LIN {X 0,Y 467.56,Z 130.239,A -85,B 0,C 180,E1 -7430.853,E2 -7430.853} C_VEL
LIN {X 0,Y 467.558,Z 130.24,A -85,B 0,C 180,E1 -7434.261,E2 -7434.261} C_VEL
LIN {X 0,Y 467.578,Z 130.242,A -85,B 0,C 180,E1 -7437.321,E2 -7437.321} C_VEL
LIN {X 0,Y 467.568,Z 130.238,A -85,B 0,C 180,E1 -7440.667,E2 -7440.667} C_VEL
LIN {X 0,Y 467.616,Z 130.238,A -85,B 0,C 180,E1 -7443.199,E2 -7443.199} C_VEL
LIN {X 0,Y 467.592,Z 130.235,A -85,B 0,C 180,E1 -7446.468,E2 -7446.468} C_VEL
LIN {X 0,Y 467.621,Z 130.233,A -85,B 0,C 180,E1 -7449.777,E2 -7449.777} C_VEL
LIN {X 0,Y 467.597,Z 130.235,A -85,B 0,C 180,E1 -7452.506,E2 -7452.506} C_VEL
LIN {X 0,Y 467.606,Z 130.241,A -85,B 0,C 180,E1 -7455.196,E2 -7455.196} C_VEL
LIN {X 0,Y 467.655,Z 130.228,A -85,B 0,C 180,E1 -7457.854,E2 -7457.854} C_VEL
LIN {X 0,Y 467.68,Z 130.228,A -85,B 0,C 180,E1 -7461.357,E2 -7461.357} C_VEL
LIN {X 0,Y 467.734,Z 130.217,A -85,B 0,C 180,E1 -7463.962,E2 -7463.962} C_VEL
LIN {X 0,Y 467.859,Z 130.204,A -85,B 0,C 180,E1 -7467.417,E2 -7467.417} C_VEL
LIN {X 0,Y 467.882,Z 130.199,A -85,B 0,C 180,E1 -7470,E2 -7470} C_VEL
LIN {X 0,Y 467.858,Z 130.208,A -85,B 0,C 180,E1 -7472.583,E2 -7472.583} C_VEL
LIN {X 0,Y 467.734,Z 130.218,A -85,B 0,C 180,E1 -7476.037,E2 -7476.037} C_VEL
LIN {X 0,Y 467.68,Z 130.232,A -85,B 0,C 180,E1 -7478.642,E2 -7478.642} C_VEL
LIN {X 0,Y 467.654,Z 130.23,A -85,B 0,C 180,E1 -7482.145,E2 -7482.145} C_VEL
LIN {X 0,Y 467.637,Z 130.23,A -85,B 0,C 180,E1 -7485.695,E2 -7485.695} C_VEL
LIN {X 0,Y 467.615,Z 130.236,A -85,B 0,C 180,E1 -7488.764,E2 -7488.764} C_VEL
LIN {X 0,Y 467.578,Z 130.237,A -85,B 0,C 180,E1 -7491.268,E2 -7491.268} C_VEL
LIN {X 0,Y 467.56,Z 130.243,A -85,B 0,C 180,E1 -7493.944,E2 -7493.944} C_VEL
LIN {X 0,Y 467.61,Z 130.234,A -85,B 0,C 180,E1 -7496.8,E2 -7496.8} C_VEL
LIN {X 0,Y 467.584,Z 130.239,A -85,B 0,C 180,E1 -7499.736,E2 -7499.736} C_VEL
LIN {X 0,Y 467.581,Z 130.238,A -85,B 0,C 180,E1 -7502.758,E2 -7502.758} C_VEL
LIN {X 0,Y 467.553,Z 130.246,A -85,B 0,C 180,E1 -7505.889,E2 -7505.889} C_VEL
LIN {X 0,Y 467.579,Z 130.237,A -85,B 0,C 180,E1 -7509.145,E2 -7509.145} C_VEL
LIN {X 0,Y 467.616,Z 130.233,A -85,B 0,C 180,E1 -7512.571,E2 -7512.571} C_VEL
LIN {X 0,Y 467.567,Z 130.239,A -85,B 0,C 180,E1 -7515.053,E2 -7515.053} C_VEL
LIN {X 0,Y 467.585,Z 130.24,A -85,B 0,C 180,E1 -7517.44,E2 -7517.44} C_VEL
LIN {X 0,Y 467.596,Z 130.235,A -85,B 0,C 180,E1 -7520.857,E2 -7520.857} C_VEL
LIN {X 0,Y 467.556,Z 130.241,A -85,B 0,C 180,E1 -7524.261,E2 -7524.261} C_VEL
LIN {X 0,Y 467.579,Z 130.241,A -85,B 0,C 180,E1 -7527.321,E2 -7527.321} C_VEL
LIN {X 0,Y 467.567,Z 130.238,A -85,B 0,C 180,E1 -7530.667,E2 -7530.667} C_VEL
LIN {X 0,Y 467.614,Z 130.237,A -85,B 0,C 180,E1 -7533.2,E2 -7533.2} C_VEL
LIN {X 0,Y 467.589,Z 130.236,A -85,B 0,C 180,E1 -7536.468,E2 -7536.468} C_VEL
LIN {X 0,Y 467.621,Z 130.234,A -85,B 0,C 180,E1 -7539.777,E2 -7539.777} C_VEL
LIN {X 0,Y 467.606,Z 130.234,A -85,B 0,C 180,E1 -7542.507,E2 -7542.507} C_VEL
LIN {X 0,Y 467.604,Z 130.242,A -85,B 0,C 180,E1 -7545.197,E2 -7545.197} C_VEL
LIN {X 0,Y 467.653,Z 130.228,A -85,B 0,C 180,E1 -7547.855,E2 -7547.855} C_VEL
LIN {X 0,Y 467.679,Z 130.228,A -85,B 0,C 180,E1 -7551.358,E2 -7551.358} C_VEL
LIN {X 0,Y 467.733,Z 130.218,A -85,B 0,C 180,E1 -7553.963,E2 -7553.963} C_VEL
LIN {X 0,Y 467.858,Z 130.204,A -85,B 0,C 180,E1 -7557.417,E2 -7557.417} C_VEL
LIN {X 0,Y 467.881,Z 130.199,A -85,B 0,C 180,E1 -7560,E2 -7560} C_VEL
LIN {X 0,Y 467.858,Z 130.207,A -85,B 0,C 180,E1 -7562.583,E2 -7562.583} C_VEL
LIN {X 0,Y 467.744,Z 130.217,A -85,B 0,C 180,E1 -7566.038,E2 -7566.038} C_VEL
LIN {X 0,Y 467.68,Z 130.232,A -85,B 0,C 180,E1 -7568.643,E2 -7568.643} C_VEL
LIN {X 0,Y 467.654,Z 130.23,A -85,B 0,C 180,E1 -7572.146,E2 -7572.146} C_VEL
LIN {X 0,Y 467.638,Z 130.23,A -85,B 0,C 180,E1 -7575.695,E2 -7575.695} C_VEL
LIN {X 0,Y 467.617,Z 130.236,A -85,B 0,C 180,E1 -7578.765,E2 -7578.765} C_VEL
LIN {X 0,Y 467.579,Z 130.237,A -85,B 0,C 180,E1 -7581.269,E2 -7581.269} C_VEL
LIN {X 0,Y 467.562,Z 130.242,A -85,B 0,C 180,E1 -7583.944,E2 -7583.944} C_VEL
LIN {X 0,Y 467.612,Z 130.235,A -85,B 0,C 180,E1 -7586.801,E2 -7586.801} C_VEL
LIN {X 0,Y 467.553,Z 130.242,A -85,B 0,C 180,E1 -7589.739,E2 -7589.739} C_VEL
LIN {X 0,Y 467.582,Z 130.238,A -85,B 0,C 180,E1 -7592.759,E2 -7592.759} C_VEL
LIN {X 0,Y 467.553,Z 130.245,A -85,B 0,C 180,E1 -7595.89,E2 -7595.89} C_VEL
LIN {X 0,Y 467.599,Z 130.234,A -85,B 0,C 180,E1 -7599.143,E2 -7599.143} C_VEL
LIN {X 0,Y 467.586,Z 130.237,A -85,B 0,C 180,E1 -7602.567,E2 -7602.567} C_VEL
LIN {X 0,Y 467.57,Z 130.238,A -85,B 0,C 180,E1 -7605.054,E2 -7605.054} C_VEL
LIN {X 0,Y 467.589,Z 130.238,A -85,B 0,C 180,E1 -7607.44,E2 -7607.44} C_VEL
LIN {X 0,Y 467.583,Z 130.236,A -85,B 0,C 180,E1 -7610.856,E2 -7610.856} C_VEL
LIN {X 0,Y 467.56,Z 130.241,A -85,B 0,C 180,E1 -7614.261,E2 -7614.261} C_VEL
LIN {X 0,Y 467.583,Z 130.24,A -85,B 0,C 180,E1 -7617.321,E2 -7617.321} C_VEL
LIN {X 0,Y 467.571,Z 130.239,A -85,B 0,C 180,E1 -7620.668,E2 -7620.668} C_VEL
LIN {X 0,Y 467.68,Z 130.252,A -85,B 0,C 180,E1 -7623.036,E2 -7623.036} C_VEL
LIN {X 0,Y 470.044,Z 142.535,A -85,B 0,C 180,E1 -7625.251,E2 -7625.251} C_VEL
LIN {X 0,Y 469.607,Z 155.018,A -85,B 0,C 180,E1 -7627.334,E2 -7627.334} C_VEL
LIN {X 0,Y 468.864,Z 174.362,A -85,B 0,C 180,E1 -7630.518,E2 -7630.518} C_VEL
LIN {X 0,Y 468.265,Z 190.123,A -85,B 0,C 180,E1 -7633.038,E2 -7633.038} C_VEL
LIN {X 0,Y 470.986,Z 210.09,A -85,B 0,C 180,E1 -7633.469,E2 -7633.469} C_VEL
LIN {X 0,Y 470.185,Z 299.083,A -85,B 0,C 180,E1 -7634.948,E2 -7634.948} C_VEL
LIN {X 0,Y 469.767,Z 311.954,A -85,B 0,C 180,E1 -7635.322,E2 -7635.322} C_VEL
LIN {X 0,Y 469.341,Z 324.553,A -85,B 0,C 180,E1 -7635.862,E2 -7635.862} C_VEL
LIN {X 0,Y 468.828,Z 336.62,A -85,B 0,C 180,E1 -7636.565,E2 -7636.565} C_VEL
LIN {X 0,Y 468.36,Z 347.957,A -85,B 0,C 180,E1 -7637.415,E2 -7637.415} C_VEL
LIN {X 0,Y 467.946,Z 358.612,A -85,B 0,C 180,E1 -7638.412,E2 -7638.412} C_VEL
LIN {X 0,Y 467.549,Z 367.139,A -85,B 0,C 180,E1 -7639.39,E2 -7639.39} C_VEL
LIN {X 0,Y 467.186,Z 376.379,A -85,B 0,C 180,E1 -7640.694,E2 -7640.694} C_VEL
LIN {X 0,Y 466.953,Z 383.82,A -85,B 0,C 180,E1 -7641.998,E2 -7641.998} C_VEL
LIN {X 0,Y 466.776,Z 389.92,A -85,B 0,C 180,E1 -7643.334,E2 -7643.334} C_VEL
LIN {X 0,Y 466.761,Z 395.107,A -85,B 0,C 180,E1 -7644.817,E2 -7644.817} C_VEL
LIN {X 0,Y 466.66,Z 397.46,A -85,B 0,C 180,E1 -7645.682,E2 -7645.682} C_VEL
LIN {X 0,Y 466.747,Z 399.385,A -85,B 0,C 180,E1 -7646.547,E2 -7646.547} C_VEL
LIN {X 0,Y 466.711,Z 400.833,A -85,B 0,C 180,E1 -7647.411,E2 -7647.411} C_VEL
LIN {X 0,Y 466.696,Z 401.849,A -85,B 0,C 180,E1 -7648.274,E2 -7648.274} C_VEL
LIN {X 0,Y 466.633,Z 402.462,A -85,B 0,C 180,E1 -7649.137,E2 -7649.137} C_VEL
LIN {X 0,Y 466.621,Z 402.677,A -85,B 0,C 180,E1 -7650,E2 -7650} C_VEL
LIN {X 0,Y 466.634,Z 402.447,A -85,B 0,C 180,E1 -7650.863,E2 -7650.863} C_VEL
LIN {X 0,Y 466.697,Z 401.808,A -85,B 0,C 180,E1 -7651.726,E2 -7651.726} C_VEL
LIN {X 0,Y 466.711,Z 400.765,A -85,B 0,C 180,E1 -7652.59,E2 -7652.59} C_VEL
LIN {X 0,Y 466.748,Z 399.31,A -85,B 0,C 180,E1 -7653.453,E2 -7653.453} C_VEL
LIN {X 0,Y 466.691,Z 396.254,A -85,B 0,C 180,E1 -7654.751,E2 -7654.751} C_VEL
LIN {X 0,Y 466.711,Z 392.13,A -85,B 0,C 180,E1 -7656.051,E2 -7656.051} C_VEL
LIN {X 0,Y 466.893,Z 385.791,A -85,B 0,C 180,E1 -7657.569,E2 -7657.569} C_VEL
LIN {X 0,Y 467.066,Z 378.887,A -85,B 0,C 180,E1 -7658.873,E2 -7658.873} C_VEL
LIN {X 0,Y 467.372,Z 370.326,A -85,B 0,C 180,E1 -7660.177,E2 -7660.177} C_VEL
LIN {X 0,Y 467.793,Z 361.513,A -85,B 0,C 180,E1 -7661.263,E2 -7661.263} C_VEL
LIN {X 0,Y 468.178,Z 351.631,A -85,B 0,C 180,E1 -7662.264,E2 -7662.264} C_VEL
LIN {X 0,Y 468.717,Z 339.929,A -85,B 0,C 180,E1 -7663.219,E2 -7663.219} C_VEL
LIN {X 0,Y 469.256,Z 327.977,A -85,B 0,C 180,E1 -7663.976,E2 -7663.976} C_VEL
LIN {X 0,Y 469.729,Z 315.638,A -85,B 0,C 180,E1 -7664.569,E2 -7664.569} C_VEL
LIN {X 0,Y 470.081,Z 304.036,A -85,B 0,C 180,E1 -7664.973,E2 -7664.973} C_VEL
LIN {X 0,Y 470.398,Z 290.664,A -85,B 0,C 180,E1 -7665.268,E2 -7665.268} C_VEL
LIN {X 0,Y 471.065,Z 208.796,A -85,B 0,C 180,E1 -7666.64,E2 -7666.64} C_VEL
LIN {X 0,Y 468.218,Z 188.105,A -85,B 0,C 180,E1 -7667.129,E2 -7667.129} C_VEL
LIN {X 0,Y 468.776,Z 170.52,A -85,B 0,C 180,E1 -7669.943,E2 -7669.943} C_VEL
LIN {X 0,Y 469.353,Z 153.611,A -85,B 0,C 180,E1 -7672.68,E2 -7672.68} C_VEL
LIN {X 0,Y 469.853,Z 142.026,A -85,B 0,C 180,E1 -7674.571,E2 -7674.571} C_VEL
LIN {X 0,Y 468.115,Z 132.345,A -85,B 0,C 180,E1 -7676.289,E2 -7676.289} C_VEL
LIN {X 0,Y 467.659,Z 130.236,A -85,B 0,C 180,E1 -7676.677,E2 -7676.677} C_VEL
LIN {X 0,Y 467.558,Z 130.25,A -85,B 0,C 180,E1 -7679.738,E2 -7679.738} C_VEL
LIN {X 0,Y 467.587,Z 130.241,A -85,B 0,C 180,E1 -7682.758,E2 -7682.758} C_VEL
LIN {X 0,Y 467.557,Z 130.246,A -85,B 0,C 180,E1 -7685.89,E2 -7685.89} C_VEL
LIN {X 0,Y 467.586,Z 130.239,A -85,B 0,C 180,E1 -7689.145,E2 -7689.145} C_VEL
LIN {X 0,Y 467.59,Z 130.239,A -85,B 0,C 180,E1 -7692.567,E2 -7692.567} C_VEL
LIN {X 0,Y 467.574,Z 130.239,A -85,B 0,C 180,E1 -7695.053,E2 -7695.053} C_VEL
LIN {X 0,Y 467.592,Z 130.239,A -85,B 0,C 180,E1 -7697.44,E2 -7697.44} C_VEL
LIN {X 0,Y 467.563,Z 130.237,A -85,B 0,C 180,E1 -7700.853,E2 -7700.853} C_VEL
LIN {X 0,Y 467.562,Z 130.239,A -85,B 0,C 180,E1 -7704.261,E2 -7704.261} C_VEL
LIN {X 0,Y 467.582,Z 130.241,A -85,B 0,C 180,E1 -7707.321,E2 -7707.321} C_VEL
LIN {X 0,Y 467.572,Z 130.239,A -85,B 0,C 180,E1 -7710.668,E2 -7710.668} C_VEL
LIN {X 0,Y 467.619,Z 130.24,A -85,B 0,C 180,E1 -7713.2,E2 -7713.2} C_VEL
LIN {X 0,Y 467.596,Z 130.236,A -85,B 0,C 180,E1 -7716.468,E2 -7716.468} C_VEL
LIN {X 0,Y 467.625,Z 130.232,A -85,B 0,C 180,E1 -7719.777,E2 -7719.777} C_VEL
LIN {X 0,Y 467.598,Z 130.235,A -85,B 0,C 180,E1 -7722.506,E2 -7722.506} C_VEL
LIN {X 0,Y 467.607,Z 130.24,A -85,B 0,C 180,E1 -7725.196,E2 -7725.196} C_VEL
LIN {X 0,Y 467.659,Z 130.229,A -85,B 0,C 180,E1 -7727.854,E2 -7727.854} C_VEL
LIN {X 0,Y 467.672,Z 130.23,A -85,B 0,C 180,E1 -7731.357,E2 -7731.357} C_VEL
LIN {X 0,Y 467.726,Z 130.223,A -85,B 0,C 180,E1 -7733.962,E2 -7733.962} C_VEL
LIN {X 0,Y 467.854,Z 130.207,A -85,B 0,C 180,E1 -7737.417,E2 -7737.417} C_VEL
LIN {X 0,Y 467.882,Z 130.204,A -85,B 0,C 180,E1 -7740,E2 -7740} C_VEL
LIN {X 0,Y 467.849,Z 130.212,A -85,B 0,C 180,E1 -7742.583,E2 -7742.583} C_VEL
LIN {X 0,Y 467.745,Z 130.412,A -85,B 0,C 180,E1 -7745.55,E2 -7745.55} C_VEL
LIN {X 0,Y 468.818,Z 136.804,A -85,B 0,C 180,E1 -7746.891,E2 -7746.891} C_VEL
LIN {X 0,Y 468.7,Z 142.276,A -85,B 0,C 180,E1 -7747.967,E2 -7747.967} C_VEL
LIN {X 0,Y 471.625,Z 155.299,A -85,B 0,C 180,E1 -7748.322,E2 -7748.322} C_VEL
LIN {X 0,Y 470.515,Z 249.579,A -85,B 0,C 180,E1 -7749.933,E2 -7749.933} C_VEL
LIN {X 0,Y 470.293,Z 262.757,A -85,B 0,C 180,E1 -7750.33,E2 -7750.33} C_VEL
LIN {X 0,Y 469.966,Z 275.289,A -85,B 0,C 180,E1 -7750.882,E2 -7750.882} C_VEL
LIN {X 0,Y 469.548,Z 286.536,A -85,B 0,C 180,E1 -7751.548,E2 -7751.548} C_VEL
LIN {X 0,Y 469.107,Z 298.008,A -85,B 0,C 180,E1 -7752.419,E2 -7752.419} C_VEL
LIN {X 0,Y 468.634,Z 308.741,A -85,B 0,C 180,E1 -7753.441,E2 -7753.441} C_VEL
LIN {X 0,Y 468.193,Z 318.16,A -85,B 0,C 180,E1 -7754.562,E2 -7754.562} C_VEL
LIN {X 0,Y 467.74,Z 327.381,A -85,B 0,C 180,E1 -7755.923,E2 -7755.923} C_VEL
LIN {X 0,Y 467.38,Z 334.621,A -85,B 0,C 180,E1 -7757.276,E2 -7757.276} C_VEL
LIN {X 0,Y 467.191,Z 340.255,A -85,B 0,C 180,E1 -7758.609,E2 -7758.609} C_VEL
LIN {X 0,Y 466.941,Z 345.531,A -85,B 0,C 180,E1 -7760.253,E2 -7760.253} C_VEL
LIN {X 0,Y 466.807,Z 347.716,A -85,B 0,C 180,E1 -7761.182,E2 -7761.182} C_VEL
LIN {X 0,Y 466.743,Z 349.422,A -85,B 0,C 180,E1 -7762.113,E2 -7762.113} C_VEL
LIN {X 0,Y 466.642,Z 350.841,A -85,B 0,C 180,E1 -7763.262,E2 -7763.262} C_VEL
LIN {X 0,Y 466.627,Z 351.641,A -85,B 0,C 180,E1 -7764.943,E2 -7764.943} C_VEL
LIN {X 0,Y 466.614,Z 351.391,A -85,B 0,C 180,E1 -7765.899,E2 -7765.899} C_VEL
LIN {X 0,Y 466.681,Z 350.122,A -85,B 0,C 180,E1 -7767.313,E2 -7767.313} C_VEL
LIN {X 0,Y 466.781,Z 347.585,A -85,B 0,C 180,E1 -7768.803,E2 -7768.803} C_VEL
LIN {X 0,Y 466.944,Z 343.795,A -85,B 0,C 180,E1 -7770.279,E2 -7770.279} C_VEL
LIN {X 0,Y 467.133,Z 338.511,A -85,B 0,C 180,E1 -7771.774,E2 -7771.774} C_VEL
LIN {X 0,Y 467.435,Z 331.467,A -85,B 0,C 180,E1 -7773.283,E2 -7773.283} C_VEL
LIN {X 0,Y 467.75,Z 324.369,A -85,B 0,C 180,E1 -7774.496,E2 -7774.496} C_VEL
LIN {X 0,Y 468.133,Z 315.195,A -85,B 0,C 180,E1 -7775.76,E2 -7775.76} C_VEL
LIN {X 0,Y 468.563,Z 305.222,A -85,B 0,C 180,E1 -7776.867,E2 -7776.867} C_VEL
LIN {X 0,Y 468.994,Z 295.409,A -85,B 0,C 180,E1 -7777.752,E2 -7777.752} C_VEL
LIN {X 0,Y 469.356,Z 284.378,A -85,B 0,C 180,E1 -7778.556,E2 -7778.556} C_VEL
LIN {X 0,Y 469.807,Z 271.549,A -85,B 0,C 180,E1 -7779.269,E2 -7779.269} C_VEL
LIN {X 0,Y 470.074,Z 258.579,A -85,B 0,C 180,E1 -7779.798,E2 -7779.798} C_VEL
LIN {X 0,Y 470.335,Z 246.28,A -85,B 0,C 180,E1 -7780.124,E2 -7780.124} C_VEL
LIN {X 0,Y 471.138,Z 154.288,A -85,B 0,C 180,E1 -7781.647,E2 -7781.647} C_VEL
LIN {X 0,Y 470.338,Z 150.488,A -85,B 0,C 180,E1 -7781.739,E2 -7781.739} C_VEL
LIN {X 0,Y 468.998,Z 146.856,A -85,B 0,C 180,E1 -7781.886,E2 -7781.886} C_VEL
LIN {X 0,Y 466.989,Z 143.798,A -85,B 0,C 180,E1 -7782.115,E2 -7782.115} C_VEL
LIN {X 0,Y 464.111,Z 140.414,A -85,B 0,C 180,E1 -7782.524,E2 -7782.524} C_VEL
LIN {X 0,Y 461.908,Z 137.477,A -85,B 0,C 180,E1 -7783.039,E2 -7783.039} C_VEL
LIN {X 0,Y 461.431,Z 136.1,A -85,B 0,C 180,E1 -7783.329,E2 -7783.329} C_VEL
LIN {X 0,Y 460.618,Z 131.109,A -85,B 0,C 180,E1 -7784.479,E2 -7784.479} C_VEL
LIN {X 0,Y 460.532,Z 131.116,A -85,B 0,C 180,E1 -7788.397,E2 -7788.397} C_VEL
LIN {X 0,Y 460.518,Z 131.12,A -85,B 0,C 180,E1 -7791.266,E2 -7791.266} C_VEL
LIN {X 0,Y 460.507,Z 131.118,A -85,B 0,C 180,E1 -7794.554,E2 -7794.554} C_VEL
LIN {X 0,Y 460.529,Z 131.12,A -85,B 0,C 180,E1 -7797.715,E2 -7797.715} C_VEL
LIN {X 0,Y 460.538,Z 131.115,A -85,B 0,C 180,E1 -7800.769,E2 -7800.769} C_VEL
LIN {X 0,Y 460.563,Z 131.114,A -85,B 0,C 180,E1 -7803.734,E2 -7803.734} C_VEL
LIN {X 0,Y 460.545,Z 131.114,A -85,B 0,C 180,E1 -7806.624,E2 -7806.624} C_VEL
LIN {X 0,Y 460.55,Z 131.118,A -85,B 0,C 180,E1 -7809.452,E2 -7809.452} C_VEL
LIN {X 0,Y 460.548,Z 131.113,A -85,B 0,C 180,E1 -7812.229,E2 -7812.229} C_VEL
LIN {X 0,Y 460.565,Z 131.116,A -85,B 0,C 180,E1 -7814.965,E2 -7814.965} C_VEL
LIN {X 0,Y 460.61,Z 131.107,A -85,B 0,C 180,E1 -7818.559,E2 -7818.559} C_VEL
LIN {X 0,Y 460.694,Z 131.095,A -85,B 0,C 180,E1 -7822.108,E2 -7822.108} C_VEL
LIN {X 0,Y 460.693,Z 131.1,A -85,B 0,C 180,E1 -7824.748,E2 -7824.748} C_VEL
LIN {X 0,Y 460.824,Z 131.08,A -85,B 0,C 180,E1 -7827.377,E2 -7827.377} C_VEL
LIN {X 0,Y 460.852,Z 131.075,A -85,B 0,C 180,E1 -7830,E2 -7830} C_VEL
LIN {X 0,Y 460.823,Z 131.085,A -85,B 0,C 180,E1 -7832.622,E2 -7832.622} C_VEL
LIN {X 0,Y 460.7,Z 131.095,A -85,B 0,C 180,E1 -7836.13,E2 -7836.13} C_VEL
LIN {X 0,Y 460.627,Z 131.109,A -85,B 0,C 180,E1 -7838.776,E2 -7838.776} C_VEL
LIN {X 0,Y 460.611,Z 131.112,A -85,B 0,C 180,E1 -7842.445,E2 -7842.445} C_VEL
LIN {X 0,Y 460.598,Z 131.109,A -85,B 0,C 180,E1 -7845.997,E2 -7845.997} C_VEL
LIN {X 0,Y 460.569,Z 131.112,A -85,B 0,C 180,E1 -7848.902,E2 -7848.902} C_VEL
LIN {X 0,Y 460.513,Z 131.117,A -85,B 0,C 180,E1 -7851.485,E2 -7851.485} C_VEL
LIN {X 0,Y 460.528,Z 131.123,A -85,B 0,C 180,E1 -7854.333,E2 -7854.333} C_VEL
LIN {X 0,Y 460.568,Z 131.11,A -85,B 0,C 180,E1 -7857.244,E2 -7857.244} C_VEL
LIN {X 0,Y 460.524,Z 131.123,A -85,B 0,C 180,E1 -7860.239,E2 -7860.239} C_VEL
LIN {X 0,Y 460.527,Z 131.116,A -85,B 0,C 180,E1 -7863.325,E2 -7863.325} C_VEL
LIN {X 0,Y 460.475,Z 131.124,A -85,B 0,C 180,E1 -7866.529,E2 -7866.529} C_VEL
LIN {X 0,Y 460.542,Z 131.113,A -85,B 0,C 180,E1 -7868.898,E2 -7868.898} C_VEL
LIN {X 0,Y 460.543,Z 131.118,A -85,B 0,C 180,E1 -7872.179,E2 -7872.179} C_VEL
LIN {X 0,Y 460.514,Z 131.12,A -85,B 0,C 180,E1 -7875.412,E2 -7875.412} C_VEL
LIN {X 0,Y 460.532,Z 131.116,A -85,B 0,C 180,E1 -7878.397,E2 -7878.397} C_VEL
LIN {X 0,Y 460.536,Z 131.117,A -85,B 0,C 180,E1 -7881.268,E2 -7881.268} C_VEL
LIN {X 0,Y 460.507,Z 131.118,A -85,B 0,C 180,E1 -7884.554,E2 -7884.554} C_VEL
LIN {X 0,Y 460.529,Z 131.121,A -85,B 0,C 180,E1 -7887.716,E2 -7887.716} C_VEL
LIN {X 0,Y 460.537,Z 131.115,A -85,B 0,C 180,E1 -7890.769,E2 -7890.769} C_VEL
LIN {X 0,Y 460.56,Z 131.115,A -85,B 0,C 180,E1 -7893.735,E2 -7893.735} C_VEL
LIN {X 0,Y 460.543,Z 131.114,A -85,B 0,C 180,E1 -7896.624,E2 -7896.624} C_VEL
LIN {X 0,Y 460.55,Z 131.119,A -85,B 0,C 180,E1 -7899.453,E2 -7899.453} C_VEL
LIN {X 0,Y 460.556,Z 131.112,A -85,B 0,C 180,E1 -7902.23,E2 -7902.23} C_VEL
LIN {X 0,Y 460.563,Z 131.116,A -85,B 0,C 180,E1 -7904.965,E2 -7904.965} C_VEL
LIN {X 0,Y 460.609,Z 131.107,A -85,B 0,C 180,E1 -7908.56,E2 -7908.56} C_VEL
LIN {X 0,Y 460.693,Z 131.095,A -85,B 0,C 180,E1 -7912.109,E2 -7912.109} C_VEL
LIN {X 0,Y 460.692,Z 131.099,A -85,B 0,C 180,E1 -7914.749,E2 -7914.749} C_VEL
LIN {X 0,Y 460.823,Z 131.081,A -85,B 0,C 180,E1 -7917.378,E2 -7917.378} C_VEL
LIN {X 0,Y 460.852,Z 131.075,A -85,B 0,C 180,E1 -7920,E2 -7920} C_VEL
LIN {X 0,Y 460.823,Z 131.084,A -85,B 0,C 180,E1 -7922.623,E2 -7922.623} C_VEL
LIN {X 0,Y 460.71,Z 131.094,A -85,B 0,C 180,E1 -7926.13,E2 -7926.13} C_VEL
LIN {X 0,Y 460.627,Z 131.11,A -85,B 0,C 180,E1 -7928.776,E2 -7928.776} C_VEL
LIN {X 0,Y 460.612,Z 131.111,A -85,B 0,C 180,E1 -7932.445,E2 -7932.445} C_VEL
LIN {X 0,Y 460.599,Z 131.108,A -85,B 0,C 180,E1 -7935.998,E2 -7935.998} C_VEL
LIN {X 0,Y 460.57,Z 131.113,A -85,B 0,C 180,E1 -7938.902,E2 -7938.902} C_VEL
LIN {X 0,Y 460.514,Z 131.117,A -85,B 0,C 180,E1 -7941.486,E2 -7941.486} C_VEL
LIN {X 0,Y 460.53,Z 131.123,A -85,B 0,C 180,E1 -7944.333,E2 -7944.333} C_VEL
LIN {X 0,Y 460.57,Z 131.11,A -85,B 0,C 180,E1 -7947.244,E2 -7947.244} C_VEL
LIN {X 0,Y 460.51,Z 131.125,A -85,B 0,C 180,E1 -7950.24,E2 -7950.24} C_VEL
LIN {X 0,Y 460.528,Z 131.115,A -85,B 0,C 180,E1 -7953.325,E2 -7953.325} C_VEL
LIN {X 0,Y 460.476,Z 131.124,A -85,B 0,C 180,E1 -7956.53,E2 -7956.53} C_VEL
LIN {X 0,Y 460.573,Z 131.115,A -85,B 0,C 180,E1 -7959.858,E2 -7959.858} C_VEL
LIN {X 0,Y 460.513,Z 131.117,A -85,B 0,C 180,E1 -7962.901,E2 -7962.901} C_VEL
LIN {X 0,Y 460.512,Z 131.125,A -85,B 0,C 180,E1 -7965.831,E2 -7965.831} C_VEL
LIN {X 0,Y 460.532,Z 131.115,A -85,B 0,C 180,E1 -7968.989,E2 -7968.989} C_VEL
LIN {X 0,Y 460.527,Z 131.117,A -85,B 0,C 180,E1 -7971.268,E2 -7971.268} C_VEL
LIN {X 0,Y 460.511,Z 131.117,A -85,B 0,C 180,E1 -7974.555,E2 -7974.555} C_VEL
LIN {X 0,Y 460.532,Z 131.122,A -85,B 0,C 180,E1 -7977.716,E2 -7977.716} C_VEL
LIN {X 0,Y 460.541,Z 131.115,A -85,B 0,C 180,E1 -7980.77,E2 -7980.77} C_VEL
LIN {X 0,Y 460.656,Z 131.258,A -85,B 0,C 180,E1 -7982.854,E2 -7982.854} C_VEL
LIN {X 0,Y 463.02,Z 143.289,A -85,B 0,C 180,E1 -7985.061,E2 -7985.061} C_VEL
LIN {X 0,Y 462.905,Z 150.398,A -85,B 0,C 180,E1 -7986.276,E2 -7986.276} C_VEL
LIN {X 0,Y 462.115,Z 167.01,A -85,B 0,C 180,E1 -7989.06,E2 -7989.06} C_VEL
LIN {X 0,Y 461.54,Z 182.195,A -85,B 0,C 180,E1 -7991.581,E2 -7991.581} C_VEL
LIN {X 0,Y 461.27,Z 189.694,A -85,B 0,C 180,E1 -7992.788,E2 -7992.788} C_VEL
LIN {X 0,Y 464.139,Z 211.478,A -85,B 0,C 180,E1 -7993.264,E2 -7993.264} C_VEL
LIN {X 0,Y 463.273,Z 298.749,A -85,B 0,C 180,E1 -7994.746,E2 -7994.746} C_VEL
LIN {X 0,Y 462.829,Z 312.351,A -85,B 0,C 180,E1 -7995.153,E2 -7995.153} C_VEL
LIN {X 0,Y 462.388,Z 324.74,A -85,B 0,C 180,E1 -7995.701,E2 -7995.701} C_VEL
LIN {X 0,Y 461.856,Z 335.858,A -85,B 0,C 180,E1 -7996.358,E2 -7996.358} C_VEL
LIN {X 0,Y 461.365,Z 347.272,A -85,B 0,C 180,E1 -7997.221,E2 -7997.221} C_VEL
LIN {X 0,Y 460.931,Z 357.99,A -85,B 0,C 180,E1 -7998.233,E2 -7998.233} C_VEL
LIN {X 0,Y 460.543,Z 366.573,A -85,B 0,C 180,E1 -7999.226,E2 -7999.226} C_VEL
LIN {X 0,Y 460.14,Z 375.862,A -85,B 0,C 180,E1 -8000.55,E2 -8000.55} C_VEL
LIN {X 0,Y 459.893,Z 383.333,A -85,B 0,C 180,E1 -8001.874,E2 -8001.874} C_VEL
LIN {X 0,Y 459.71,Z 389.715,A -85,B 0,C 180,E1 -8003.295,E2 -8003.295} C_VEL
LIN {X 0,Y 459.669,Z 394.672,A -85,B 0,C 180,E1 -8004.737,E2 -8004.737} C_VEL
LIN {X 0,Y 459.575,Z 397.035,A -85,B 0,C 180,E1 -8005.615,E2 -8005.615} C_VEL
LIN {X 0,Y 459.657,Z 398.967,A -85,B 0,C 180,E1 -8006.494,E2 -8006.494} C_VEL
LIN {X 0,Y 459.631,Z 400.429,A -85,B 0,C 180,E1 -8007.371,E2 -8007.371} C_VEL
LIN {X 0,Y 459.633,Z 401.451,A -85,B 0,C 180,E1 -8008.248,E2 -8008.248} C_VEL
LIN {X 0,Y 459.566,Z 402.068,A -85,B 0,C 180,E1 -8009.124,E2 -8009.124} C_VEL
LIN {X 0,Y 459.551,Z 402.287,A -85,B 0,C 180,E1 -8010,E2 -8010} C_VEL
LIN {X 0,Y 459.566,Z 402.062,A -85,B 0,C 180,E1 -8010.877,E2 -8010.877} C_VEL
LIN {X 0,Y 459.604,Z 401.422,A -85,B 0,C 180,E1 -8011.753,E2 -8011.753} C_VEL
LIN {X 0,Y 459.631,Z 400.38,A -85,B 0,C 180,E1 -8012.629,E2 -8012.629} C_VEL
LIN {X 0,Y 459.642,Z 398.925,A -85,B 0,C 180,E1 -8013.507,E2 -8013.507} C_VEL
LIN {X 0,Y 459.622,Z 395.872,A -85,B 0,C 180,E1 -8014.825,E2 -8014.825} C_VEL
LIN {X 0,Y 459.636,Z 391.015,A -85,B 0,C 180,E1 -8016.343,E2 -8016.343} C_VEL
LIN {X 0,Y 459.864,Z 384.372,A -85,B 0,C 180,E1 -8017.906,E2 -8017.906} C_VEL
LIN {X 0,Y 460.073,Z 377.228,A -85,B 0,C 180,E1 -8019.23,E2 -8019.23} C_VEL
LIN {X 0,Y 460.418,Z 368.282,A -85,B 0,C 180,E1 -8020.555,E2 -8020.555} C_VEL
LIN {X 0,Y 460.923,Z 358.149,A -85,B 0,C 180,E1 -8021.768,E2 -8021.768} C_VEL
LIN {X 0,Y 461.323,Z 347.946,A -85,B 0,C 180,E1 -8022.754,E2 -8022.754} C_VEL
LIN {X 0,Y 461.924,Z 336.447,A -85,B 0,C 180,E1 -8023.641,E2 -8023.641} C_VEL
LIN {X 0,Y 462.497,Z 323.667,A -85,B 0,C 180,E1 -8024.409,E2 -8024.409} C_VEL
LIN {X 0,Y 463.011,Z 310.491,A -85,B 0,C 180,E1 -8024.982,E2 -8024.982} C_VEL
LIN {X 0,Y 463.461,Z 297.658,A -85,B 0,C 180,E1 -8025.361,E2 -8025.361} C_VEL
LIN {X 0,Y 464.326,Z 209.748,A -85,B 0,C 180,E1 -8026.889,E2 -8026.889} C_VEL
LIN {X 0,Y 461.265,Z 187.591,A -85,B 0,C 180,E1 -8027.433,E2 -8027.433} C_VEL
LIN {X 0,Y 461.808,Z 171.671,A -85,B 0,C 180,E1 -8030.024,E2 -8030.024} C_VEL
LIN {X 0,Y 462.516,Z 153.338,A -85,B 0,C 180,E1 -8033.034,E2 -8033.034} C_VEL
LIN {X 0,Y 462.958,Z 143.377,A -85,B 0,C 180,E1 -8034.691,E2 -8034.691} C_VEL
LIN {X 0,Y 460.841,Z 132.118,A -85,B 0,C 180,E1 -8036.737,E2 -8036.737} C_VEL
LIN {X 0,Y 460.628,Z 131.112,A -85,B 0,C 180,E1 -8036.934,E2 -8036.934} C_VEL
LIN {X 0,Y 460.514,Z 131.129,A -85,B 0,C 180,E1 -8040.24,E2 -8040.24} C_VEL
LIN {X 0,Y 460.533,Z 131.117,A -85,B 0,C 180,E1 -8043.325,E2 -8043.325} C_VEL
LIN {X 0,Y 460.48,Z 131.126,A -85,B 0,C 180,E1 -8046.529,E2 -8046.529} C_VEL
LIN {X 0,Y 460.561,Z 131.119,A -85,B 0,C 180,E1 -8049.86,E2 -8049.86} C_VEL
LIN {X 0,Y 460.517,Z 131.119,A -85,B 0,C 180,E1 -8052.9,E2 -8052.9} C_VEL
LIN {X 0,Y 460.515,Z 131.122,A -85,B 0,C 180,E1 -8055.83,E2 -8055.83} C_VEL
LIN {X 0,Y 460.534,Z 131.113,A -85,B 0,C 180,E1 -8058.989,E2 -8058.989} C_VEL
LIN {X 0,Y 460.522,Z 131.116,A -85,B 0,C 180,E1 -8061.266,E2 -8061.266} C_VEL
LIN {X 0,Y 460.511,Z 131.117,A -85,B 0,C 180,E1 -8064.554,E2 -8064.554} C_VEL
LIN {X 0,Y 460.533,Z 131.117,A -85,B 0,C 180,E1 -8067.715,E2 -8067.715} C_VEL
LIN {X 0,Y 460.542,Z 131.116,A -85,B 0,C 180,E1 -8070.769,E2 -8070.769} C_VEL
LIN {X 0,Y 460.562,Z 131.112,A -85,B 0,C 180,E1 -8073.734,E2 -8073.734} C_VEL
LIN {X 0,Y 460.549,Z 131.115,A -85,B 0,C 180,E1 -8076.624,E2 -8076.624} C_VEL
LIN {X 0,Y 460.554,Z 131.115,A -85,B 0,C 180,E1 -8079.453,E2 -8079.453} C_VEL
LIN {X 0,Y 460.549,Z 131.111,A -85,B 0,C 180,E1 -8082.229,E2 -8082.229} C_VEL
LIN {X 0,Y 460.567,Z 131.116,A -85,B 0,C 180,E1 -8084.965,E2 -8084.965} C_VEL
LIN {X 0,Y 460.613,Z 131.111,A -85,B 0,C 180,E1 -8088.559,E2 -8088.559} C_VEL
LIN {X 0,Y 460.622,Z 131.11,A -85,B 0,C 180,E1 -8091.223,E2 -8091.223} C_VEL
LIN {X 0,Y 460.69,Z 131.1,A -85,B 0,C 180,E1 -8093.87,E2 -8093.87} C_VEL
LIN {X 0,Y 460.794,Z 131.087,A -85,B 0,C 180,E1 -8097.377,E2 -8097.377} C_VEL
LIN {X 0,Y 460.852,Z 131.08,A -85,B 0,C 180,E1 -8100,E2 -8100} C_VEL
LIN {X 0,Y 460.789,Z 131.091,A -85,B 0,C 180,E1 -8102.622,E2 -8102.622} C_VEL
LIN {X 0,Y 460.723,Z 131.294,A -85,B 0,C 180,E1 -8105.306,E2 -8105.306} C_VEL
LIN {X 0,Y 461.923,Z 138.182,A -85,B 0,C 180,E1 -8106.771,E2 -8106.771} C_VEL
LIN {X 0,Y 461.855,Z 142.893,A -85,B 0,C 180,E1 -8107.679,E2 -8107.679} C_VEL
LIN {X 0,Y 464.829,Z 155.977,A -85,B 0,C 180,E1 -8108.051,E2 -8108.051} C_VEL
LIN {X 0,Y 463.722,Z 250.279,A -85,B 0,C 180,E1 -8109.702,E2 -8109.702} C_VEL
LIN {X 0,Y 463.464,Z 263.35,A -85,B 0,C 180,E1 -8110.105,E2 -8110.105} C_VEL
LIN {X 0,Y 463.129,Z 275.663,A -85,B 0,C 180,E1 -8110.658,E2 -8110.658} C_VEL
LIN {X 0,Y 462.643,Z 287.723,A -85,B 0,C 180,E1 -8111.389,E2 -8111.389} C_VEL
LIN {X 0,Y 462.165,Z 299.258,A -85,B 0,C 180,E1 -8112.292,E2 -8112.292} C_VEL
LIN {X 0,Y 461.687,Z 309.646,A -85,B 0,C 180,E1 -8113.311,E2 -8113.311} C_VEL
LIN {X 0,Y 461.155,Z 319.83,A -85,B 0,C 180,E1 -8114.564,E2 -8114.564} C_VEL
LIN {X 0,Y 460.782,Z 327.374,A -85,B 0,C 180,E1 -8115.707,E2 -8115.707} C_VEL
LIN {X 0,Y 460.365,Z 334.764,A -85,B 0,C 180,E1 -8117.09,E2 -8117.09} C_VEL
LIN {X 0,Y 460.149,Z 339.73,A -85,B 0,C 180,E1 -8118.246,E2 -8118.246} C_VEL
LIN {X 0,Y 459.946,Z 344.458,A -85,B 0,C 180,E1 -8119.643,E2 -8119.643} C_VEL
LIN {X 0,Y 459.737,Z 348.237,A -85,B 0,C 180,E1 -8121.171,E2 -8121.171} C_VEL
LIN {X 0,Y 459.615,Z 350.413,A -85,B 0,C 180,E1 -8122.474,E2 -8122.474} C_VEL
LIN {X 0,Y 459.569,Z 351.421,A -85,B 0,C 180,E1 -8123.428,E2 -8123.428} C_VEL
LIN {X 0,Y 459.529,Z 351.956,A -85,B 0,C 180,E1 -8124.389,E2 -8124.389} C_VEL
LIN {X 0,Y 459.528,Z 351.931,A -85,B 0,C 180,E1 -8125.532,E2 -8125.532} C_VEL
LIN {X 0,Y 459.563,Z 351.526,A -85,B 0,C 180,E1 -8126.326,E2 -8126.326} C_VEL
LIN {X 0,Y 459.594,Z 350.27,A -85,B 0,C 180,E1 -8127.511,E2 -8127.511} C_VEL
LIN {X 0,Y 459.695,Z 348.077,A -85,B 0,C 180,E1 -8128.789,E2 -8128.789} C_VEL
LIN {X 0,Y 459.885,Z 344.324,A -85,B 0,C 180,E1 -8130.285,E2 -8130.285} C_VEL
LIN {X 0,Y 460.084,Z 339.097,A -85,B 0,C 180,E1 -8131.803,E2 -8131.803} C_VEL
LIN {X 0,Y 460.375,Z 332.086,A -85,B 0,C 180,E1 -8133.337,E2 -8133.337} C_VEL
LIN {X 0,Y 460.753,Z 324.373,A -85,B 0,C 180,E1 -8134.672,E2 -8134.672} C_VEL
LIN {X 0,Y 461.116,Z 315.622,A -85,B 0,C 180,E1 -8135.89,E2 -8135.89} C_VEL
LIN {X 0,Y 461.564,Z 306.034,A -85,B 0,C 180,E1 -8136.973,E2 -8136.973} C_VEL
LIN {X 0,Y 462.076,Z 295.117,A -85,B 0,C 180,E1 -8137.971,E2 -8137.971} C_VEL
LIN {X 0,Y 462.453,Z 283.852,A -85,B 0,C 180,E1 -8138.788,E2 -8138.788} C_VEL
LIN {X 0,Y 462.919,Z 271.089,A -85,B 0,C 180,E1 -8139.496,E2 -8139.496} C_VEL
LIN {X 0,Y 463.196,Z 258.353,A -85,B 0,C 180,E1 -8140.012,E2 -8140.012} C_VEL
LIN {X 0,Y 463.465,Z 244.926,A -85,B 0,C 180,E1 -8140.357,E2 -8140.357} C_VEL
LIN {X 0,Y 464.327,Z 155.469,A -85,B 0,C 180,E1 -8141.861,E2 -8141.861} C_VEL
LIN {X 0,Y 461.466,Z 141.223,A -85,B 0,C 180,E1 -8142.236,E2 -8142.236} C_VEL
LIN {X 0,Y 461.431,Z 136.1,A -85,B 0,C 180,E1 -8143.329,E2 -8143.329} C_VEL
LIN {X 0,Y 460.498,Z 134.417,A -85,B 0,C 180,E1 -8143.766,E2 -8143.766} C_VEL
LIN {X 0,Y 458.694,Z 133.265,A -85,B 0,C 180,E1 -8144.199,E2 -8144.199} C_VEL
LIN {X 0,Y 454.707,Z 132.159,A -85,B 0,C 180,E1 -8145.09,E2 -8145.09} C_VEL
LIN {X 0,Y 453.5,Z 132.003,A -85,B 0,C 180,E1 -8145.665,E2 -8145.665} C_VEL
LIN {X 0,Y 453.472,Z 132.002,A -85,B 0,C 180,E1 -8145.75,E2 -8145.75} C_VEL
LIN {X 0,Y 453.479,Z 131.996,A -85,B 0,C 180,E1 -8148.209,E2 -8148.209} C_VEL
LIN {X 0,Y 453.487,Z 131.992,A -85,B 0,C 180,E1 -8150.794,E2 -8150.794} C_VEL
LIN {X 0,Y 453.453,Z 132,A -85,B 0,C 180,E1 -8153.917,E2 -8153.917} C_VEL
LIN {X 0,Y 453.478,Z 131.997,A -85,B 0,C 180,E1 -8157.15,E2 -8157.15} C_VEL
LIN {X 0,Y 453.473,Z 131.994,A -85,B 0,C 180,E1 -8160.268,E2 -8160.268} C_VEL
LIN {X 0,Y 453.506,Z 131.997,A -85,B 0,C 180,E1 -8163.294,E2 -8163.294} C_VEL
LIN {X 0,Y 453.502,Z 131.99,A -85,B 0,C 180,E1 -8166.238,E2 -8166.238} C_VEL
LIN {X 0,Y 453.482,Z 131.999,A -85,B 0,C 180,E1 -8169.117,E2 -8169.117} C_VEL
LIN {X 0,Y 453.502,Z 131.991,A -85,B 0,C 180,E1 -8171.944,E2 -8171.944} C_VEL
LIN {X 0,Y 453.539,Z 131.989,A -85,B 0,C 180,E1 -8174.726,E2 -8174.726} C_VEL
LIN {X 0,Y 453.559,Z 131.984,A -85,B 0,C 180,E1 -8178.379,E2 -8178.379} C_VEL
LIN {X 0,Y 453.651,Z 131.972,A -85,B 0,C 180,E1 -8181.985,E2 -8181.985} C_VEL
LIN {X 0,Y 453.666,Z 131.974,A -85,B 0,C 180,E1 -8184.666,E2 -8184.666} C_VEL
LIN {X 0,Y 453.764,Z 131.96,A -85,B 0,C 180,E1 -8187.336,E2 -8187.336} C_VEL
LIN {X 0,Y 453.823,Z 131.951,A -85,B 0,C 180,E1 -8190,E2 -8190} C_VEL
LIN {X 0,Y 453.763,Z 131.965,A -85,B 0,C 180,E1 -8192.663,E2 -8192.663} C_VEL
LIN {X 0,Y 453.668,Z 131.972,A -85,B 0,C 180,E1 -8196.225,E2 -8196.225} C_VEL
LIN {X 0,Y 453.591,Z 131.983,A -85,B 0,C 180,E1 -8198.913,E2 -8198.913} C_VEL
LIN {X 0,Y 453.561,Z 131.991,A -85,B 0,C 180,E1 -8202.529,E2 -8202.529} C_VEL
LIN {X 0,Y 453.542,Z 131.99,A -85,B 0,C 180,E1 -8206.196,E2 -8206.196} C_VEL
LIN {X 0,Y 453.518,Z 131.989,A -85,B 0,C 180,E1 -8209.041,E2 -8209.041} C_VEL
LIN {X 0,Y 453.474,Z 131.996,A -85,B 0,C 180,E1 -8211.836,E2 -8211.836} C_VEL
LIN {X 0,Y 453.498,Z 131.993,A -85,B 0,C 180,E1 -8214.735,E2 -8214.735} C_VEL
LIN {X 0,Y 453.53,Z 131.991,A -85,B 0,C 180,E1 -8217.96,E2 -8217.96} C_VEL
LIN {X 0,Y 453.48,Z 131.994,A -85,B 0,C 180,E1 -8220.759,E2 -8220.759} C_VEL
LIN {X 0,Y 453.475,Z 131.999,A -85,B 0,C 180,E1 -8223.912,E2 -8223.912} C_VEL
LIN {X 0,Y 453.467,Z 131.995,A -85,B 0,C 180,E1 -8227.188,E2 -8227.188} C_VEL
LIN {X 0,Y 453.502,Z 131.992,A -85,B 0,C 180,E1 -8229.448,E2 -8229.448} C_VEL
LIN {X 0,Y 453.489,Z 131.992,A -85,B 0,C 180,E1 -8232.991,E2 -8232.991} C_VEL
LIN {X 0,Y 453.463,Z 132.003,A -85,B 0,C 180,E1 -8235.779,E2 -8235.779} C_VEL
LIN {X 0,Y 453.513,Z 131.993,A -85,B 0,C 180,E1 -8239.406,E2 -8239.406} C_VEL
LIN {X 0,Y 453.472,Z 131.996,A -85,B 0,C 180,E1 -8242.223,E2 -8242.223} C_VEL
LIN {X 0,Y 453.484,Z 131.996,A -85,B 0,C 180,E1 -8245.223,E2 -8245.223} C_VEL
LIN {X 0,Y 453.463,Z 131.995,A -85,B 0,C 180,E1 -8248.475,E2 -8248.475} C_VEL
LIN {X 0,Y 453.529,Z 131.989,A -85,B 0,C 180,E1 -8252.04,E2 -8252.04} C_VEL
LIN {X 0,Y 453.51,Z 131.995,A -85,B 0,C 180,E1 -8255.266,E2 -8255.266} C_VEL
LIN {X 0,Y 453.477,Z 131.994,A -85,B 0,C 180,E1 -8258.415,E2 -8258.415} C_VEL
LIN {X 0,Y 453.52,Z 131.992,A -85,B 0,C 180,E1 -8261.009,E2 -8261.009} C_VEL
LIN {X 0,Y 453.566,Z 131.983,A -85,B 0,C 180,E1 -8263.88,E2 -8263.88} C_VEL
LIN {X 0,Y 453.561,Z 131.987,A -85,B 0,C 180,E1 -8267.471,E2 -8267.471} C_VEL
LIN {X 0,Y 453.59,Z 131.987,A -85,B 0,C 180,E1 -8271.087,E2 -8271.087} C_VEL
LIN {X 0,Y 453.667,Z 131.97,A -85,B 0,C 180,E1 -8273.775,E2 -8273.775} C_VEL
LIN {X 0,Y 453.763,Z 131.961,A -85,B 0,C 180,E1 -8277.337,E2 -8277.337} C_VEL
LIN {X 0,Y 453.822,Z 131.951,A -85,B 0,C 180,E1 -8280,E2 -8280} C_VEL
LIN {X 0,Y 453.763,Z 131.964,A -85,B 0,C 180,E1 -8282.664,E2 -8282.664} C_VEL
LIN {X 0,Y 453.677,Z 131.97,A -85,B 0,C 180,E1 -8286.226,E2 -8286.226} C_VEL
LIN {X 0,Y 453.591,Z 131.984,A -85,B 0,C 180,E1 -8288.914,E2 -8288.914} C_VEL
LIN {X 0,Y 453.562,Z 131.99,A -85,B 0,C 180,E1 -8292.529,E2 -8292.529} C_VEL
LIN {X 0,Y 453.543,Z 131.989,A -85,B 0,C 180,E1 -8296.196,E2 -8296.196} C_VEL
LIN {X 0,Y 453.519,Z 131.99,A -85,B 0,C 180,E1 -8299.041,E2 -8299.041} C_VEL
LIN {X 0,Y 453.475,Z 131.995,A -85,B 0,C 180,E1 -8301.837,E2 -8301.837} C_VEL
LIN {X 0,Y 453.499,Z 131.994,A -85,B 0,C 180,E1 -8304.736,E2 -8304.736} C_VEL
LIN {X 0,Y 453.531,Z 131.991,A -85,B 0,C 180,E1 -8307.96,E2 -8307.96} C_VEL
LIN {X 0,Y 453.465,Z 131.996,A -85,B 0,C 180,E1 -8311.526,E2 -8311.526} C_VEL
LIN {X 0,Y 453.487,Z 131.993,A -85,B 0,C 180,E1 -8314.778,E2 -8314.778} C_VEL
LIN {X 0,Y 453.48,Z 131.998,A -85,B 0,C 180,E1 -8318.31,E2 -8318.31} C_VEL
LIN {X 0,Y 453.516,Z 131.99,A -85,B 0,C 180,E1 -8320.607,E2 -8320.607} C_VEL
LIN {X 0,Y 453.466,Z 131.999,A -85,B 0,C 180,E1 -8324.221,E2 -8324.221} C_VEL
LIN {X 0,Y 453.463,Z 131.995,A -85,B 0,C 180,E1 -8327.006,E2 -8327.006} C_VEL
LIN {X 0,Y 453.495,Z 131.994,A -85,B 0,C 180,E1 -8329.409,E2 -8329.409} C_VEL
LIN {X 0,Y 453.451,Z 131.999,A -85,B 0,C 180,E1 -8332.228,E2 -8332.228} C_VEL
LIN {X 0,Y 453.488,Z 131.994,A -85,B 0,C 180,E1 -8335.223,E2 -8335.223} C_VEL
LIN {X 0,Y 453.467,Z 131.997,A -85,B 0,C 180,E1 -8338.475,E2 -8338.475} C_VEL
LIN {X 0,Y 453.534,Z 131.992,A -85,B 0,C 180,E1 -8342.041,E2 -8342.041} C_VEL
LIN {X 0,Y 453.609,Z 132.136,A -85,B 0,C 180,E1 -8342.647,E2 -8342.647} C_VEL
LIN {X 0,Y 456.02,Z 144.362,A -85,B 0,C 180,E1 -8344.925,E2 -8344.925} C_VEL
LIN {X 0,Y 456.049,Z 149.932,A -85,B 0,C 180,E1 -8345.897,E2 -8345.897} C_VEL
LIN {X 0,Y 455.126,Z 167.917,A -85,B 0,C 180,E1 -8348.96,E2 -8348.96} C_VEL
LIN {X 0,Y 454.528,Z 183.102,A -85,B 0,C 180,E1 -8351.52,E2 -8351.52} C_VEL
LIN {X 0,Y 454.281,Z 189.445,A -85,B 0,C 180,E1 -8352.541,E2 -8352.541} C_VEL
LIN {X 0,Y 457.283,Z 211.863,A -85,B 0,C 180,E1 -8353.042,E2 -8353.042} C_VEL
LIN {X 0,Y 456.345,Z 298.328,A -85,B 0,C 180,E1 -8354.537,E2 -8354.537} C_VEL
LIN {X 0,Y 455.922,Z 311.933,A -85,B 0,C 180,E1 -8354.951,E2 -8354.951} C_VEL
LIN {X 0,Y 455.435,Z 324.849,A -85,B 0,C 180,E1 -8355.535,E2 -8355.535} C_VEL
LIN {X 0,Y 454.829,Z 336.647,A -85,B 0,C 180,E1 -8356.257,E2 -8356.257} C_VEL
LIN {X 0,Y 454.316,Z 348.79,A -85,B 0,C 180,E1 -8357.214,E2 -8357.214} C_VEL
LIN {X 0,Y 453.866,Z 358.386,A -85,B 0,C 180,E1 -8358.161,E2 -8358.161} C_VEL
LIN {X 0,Y 453.428,Z 367.656,A -85,B 0,C 180,E1 -8359.281,E2 -8359.281} C_VEL
LIN {X 0,Y 453.023,Z 376.688,A -85,B 0,C 180,E1 -8360.626,E2 -8360.626} C_VEL
LIN {X 0,Y 452.778,Z 383.938,A -85,B 0,C 180,E1 -8361.97,E2 -8361.97} C_VEL
LIN {X 0,Y 452.604,Z 389.863,A -85,B 0,C 180,E1 -8363.357,E2 -8363.357} C_VEL
LIN {X 0,Y 452.577,Z 394.224,A -85,B 0,C 180,E1 -8364.654,E2 -8364.654} C_VEL
LIN {X 0,Y 452.496,Z 396.598,A -85,B 0,C 180,E1 -8365.546,E2 -8365.546} C_VEL
LIN {X 0,Y 452.553,Z 398.539,A -85,B 0,C 180,E1 -8366.439,E2 -8366.439} C_VEL
LIN {X 0,Y 452.554,Z 400.018,A -85,B 0,C 180,E1 -8367.33,E2 -8367.33} C_VEL
LIN {X 0,Y 452.541,Z 401.046,A -85,B 0,C 180,E1 -8368.22,E2 -8368.22} C_VEL
LIN {X 0,Y 452.501,Z 401.67,A -85,B 0,C 180,E1 -8369.11,E2 -8369.11} C_VEL
LIN {X 0,Y 452.483,Z 401.894,A -85,B 0,C 180,E1 -8370,E2 -8370} C_VEL
LIN {X 0,Y 452.501,Z 401.679,A -85,B 0,C 180,E1 -8370.89,E2 -8370.89} C_VEL
LIN {X 0,Y 452.515,Z 401.041,A -85,B 0,C 180,E1 -8371.78,E2 -8371.78} C_VEL
LIN {X 0,Y 452.553,Z 400.001,A -85,B 0,C 180,E1 -8372.671,E2 -8372.671} C_VEL
LIN {X 0,Y 452.538,Z 398.547,A -85,B 0,C 180,E1 -8373.562,E2 -8373.562} C_VEL
LIN {X 0,Y 452.552,Z 395.495,A -85,B 0,C 180,E1 -8374.9,E2 -8374.9} C_VEL
LIN {X 0,Y 452.555,Z 391.054,A -85,B 0,C 180,E1 -8376.332,E2 -8376.332} C_VEL
LIN {X 0,Y 452.742,Z 385.043,A -85,B 0,C 180,E1 -8377.807,E2 -8377.807} C_VEL
LIN {X 0,Y 452.98,Z 378.142,A -85,B 0,C 180,E1 -8379.151,E2 -8379.151} C_VEL
LIN {X 0,Y 453.333,Z 369.589,A -85,B 0,C 180,E1 -8380.496,E2 -8380.496} C_VEL
LIN {X 0,Y 453.813,Z 360.792,A -85,B 0,C 180,E1 -8381.615,E2 -8381.615} C_VEL
LIN {X 0,Y 454.224,Z 351.025,A -85,B 0,C 180,E1 -8382.638,E2 -8382.638} C_VEL
LIN {X 0,Y 454.848,Z 339.282,A -85,B 0,C 180,E1 -8383.629,E2 -8383.629} C_VEL
LIN {X 0,Y 455.464,Z 327.439,A -85,B 0,C 180,E1 -8384.408,E2 -8384.408} C_VEL
LIN {X 0,Y 455.995,Z 315.228,A -85,B 0,C 180,E1 -8385.018,E2 -8385.018} C_VEL
LIN {X 0,Y 456.449,Z 302.968,A -85,B 0,C 180,E1 -8385.46,E2 -8385.46} C_VEL
LIN {X 0,Y 456.749,Z 289.574,A -85,B 0,C 180,E1 -8385.764,E2 -8385.764} C_VEL
LIN {X 0,Y 457.556,Z 210.274,A -85,B 0,C 180,E1 -8387.156,E2 -8387.156} C_VEL
LIN {X 0,Y 454.702,Z 189.706,A -85,B 0,C 180,E1 -8387.664,E2 -8387.664} C_VEL
LIN {X 0,Y 454.291,Z 187.058,A -85,B 0,C 180,E1 -8387.758,E2 -8387.758} C_VEL
LIN {X 0,Y 454.852,Z 172.806,A -85,B 0,C 180,E1 -8390.108,E2 -8390.108} C_VEL
LIN {X 0,Y 455.615,Z 154.553,A -85,B 0,C 180,E1 -8393.163,E2 -8393.163} C_VEL
LIN {X 0,Y 456.065,Z 144.691,A -85,B 0,C 180,E1 -8394.83,E2 -8394.83} C_VEL
LIN {X 0,Y 453.885,Z 133.395,A -85,B 0,C 180,E1 -8396.931,E2 -8396.931} C_VEL
LIN {X 0,Y 453.584,Z 131.989,A -85,B 0,C 180,E1 -8397.199,E2 -8397.199} C_VEL
LIN {X 0,Y 453.48,Z 132.002,A -85,B 0,C 180,E1 -8400.76,E2 -8400.76} C_VEL
LIN {X 0,Y 453.48,Z 132,A -85,B 0,C 180,E1 -8403.913,E2 -8403.913} C_VEL
LIN {X 0,Y 453.456,Z 131.999,A -85,B 0,C 180,E1 -8407.19,E2 -8407.19} C_VEL
LIN {X 0,Y 453.52,Z 131.993,A -85,B 0,C 180,E1 -8409.447,E2 -8409.447} C_VEL
LIN {X 0,Y 453.467,Z 131.997,A -85,B 0,C 180,E1 -8412.995,E2 -8412.995} C_VEL
LIN {X 0,Y 453.47,Z 132,A -85,B 0,C 180,E1 -8415.779,E2 -8415.779} C_VEL
LIN {X 0,Y 453.483,Z 131.993,A -85,B 0,C 180,E1 -8418.209,E2 -8418.209} C_VEL
LIN {X 0,Y 453.49,Z 131.99,A -85,B 0,C 180,E1 -8420.794,E2 -8420.794} C_VEL
LIN {X 0,Y 453.457,Z 131.999,A -85,B 0,C 180,E1 -8423.917,E2 -8423.917} C_VEL
LIN {X 0,Y 453.482,Z 131.995,A -85,B 0,C 180,E1 -8427.151,E2 -8427.151} C_VEL
LIN {X 0,Y 453.477,Z 131.995,A -85,B 0,C 180,E1 -8430.268,E2 -8430.268} C_VEL
LIN {X 0,Y 453.508,Z 131.996,A -85,B 0,C 180,E1 -8433.294,E2 -8433.294} C_VEL
LIN {X 0,Y 453.505,Z 131.991,A -85,B 0,C 180,E1 -8436.239,E2 -8436.239} C_VEL
LIN {X 0,Y 453.486,Z 131.997,A -85,B 0,C 180,E1 -8439.117,E2 -8439.117} C_VEL
LIN {X 0,Y 453.504,Z 131.988,A -85,B 0,C 180,E1 -8441.944,E2 -8441.944} C_VEL
LIN {X 0,Y 453.542,Z 131.989,A -85,B 0,C 180,E1 -8444.726,E2 -8444.726} C_VEL
LIN {X 0,Y 453.562,Z 131.988,A -85,B 0,C 180,E1 -8448.379,E2 -8448.379} C_VEL
LIN {X 0,Y 453.588,Z 131.987,A -85,B 0,C 180,E1 -8451.086,E2 -8451.086} C_VEL
LIN {X 0,Y 453.655,Z 131.976,A -85,B 0,C 180,E1 -8453.774,E2 -8453.774} C_VEL
LIN {X 0,Y 453.738,Z 131.967,A -85,B 0,C 180,E1 -8457.336,E2 -8457.336} C_VEL
LIN {X 0,Y 453.822,Z 131.956,A -85,B 0,C 180,E1 -8460,E2 -8460} C_VEL
LIN {X 0,Y 453.733,Z 131.97,A -85,B 0,C 180,E1 -8462.663,E2 -8462.663} C_VEL
LIN {X 0,Y 453.625,Z 132.096,A -85,B 0,C 180,E1 -8465.027,E2 -8465.027} C_VEL
LIN {X 0,Y 455.012,Z 139.598,A -85,B 0,C 180,E1 -8466.652,E2 -8466.652} C_VEL
LIN {X 0,Y 454.964,Z 142.995,A -85,B 0,C 180,E1 -8467.349,E2 -8467.349} C_VEL
LIN {X 0,Y 458.192,Z 157.966,A -85,B 0,C 180,E1 -8467.796,E2 -8467.796} C_VEL
LIN {X 0,Y 456.915,Z 251.017,A -85,B 0,C 180,E1 -8469.461,E2 -8469.461} C_VEL
LIN {X 0,Y 456.655,Z 264.012,A -85,B 0,C 180,E1 -8469.873,E2 -8469.873} C_VEL
LIN {X 0,Y 456.281,Z 276.826,A -85,B 0,C 180,E1 -8470.466,E2 -8470.466} C_VEL
LIN {X 0,Y 455.746,Z 288.969,A -85,B 0,C 180,E1 -8471.226,E2 -8471.226} C_VEL
LIN {X 0,Y 455.244,Z 300.354,A -85,B 0,C 180,E1 -8472.142,E2 -8472.142} C_VEL
LIN {X 0,Y 454.74,Z 310.583,A -85,B 0,C 180,E1 -8473.178,E2 -8473.178} C_VEL
LIN {X 0,Y 454.224,Z 319.83,A -85,B 0,C 180,E1 -8474.333,E2 -8474.333} C_VEL
LIN {X 0,Y 453.729,Z 328.73,A -85,B 0,C 180,E1 -8475.71,E2 -8475.71} C_VEL
LIN {X 0,Y 453.323,Z 335.967,A -85,B 0,C 180,E1 -8477.131,E2 -8477.131} C_VEL
LIN {X 0,Y 453.082,Z 341.344,A -85,B 0,C 180,E1 -8478.462,E2 -8478.462} C_VEL
LIN {X 0,Y 452.838,Z 346.024,A -85,B 0,C 180,E1 -8479.964,E2 -8479.964} C_VEL
LIN {X 0,Y 452.668,Z 349.089,A -85,B 0,C 180,E1 -8481.323,E2 -8481.323} C_VEL
LIN {X 0,Y 452.512,Z 351.339,A -85,B 0,C 180,E1 -8482.847,E2 -8482.847} C_VEL
LIN {X 0,Y 452.467,Z 352.105,A -85,B 0,C 180,E1 -8483.819,E2 -8483.819} C_VEL
LIN {X 0,Y 452.426,Z 352.414,A -85,B 0,C 180,E1 -8484.798,E2 -8484.798} C_VEL
LIN {X 0,Y 452.471,Z 352.236,A -85,B 0,C 180,E1 -8485.779,E2 -8485.779} C_VEL
LIN {X 0,Y 452.474,Z 351.525,A -85,B 0,C 180,E1 -8486.771,E2 -8486.771} C_VEL
LIN {X 0,Y 452.532,Z 350.339,A -85,B 0,C 180,E1 -8487.769,E2 -8487.769} C_VEL
LIN {X 0,Y 452.606,Z 348.565,A -85,B 0,C 180,E1 -8488.774,E2 -8488.774} C_VEL
LIN {X 0,Y 452.816,Z 344.847,A -85,B 0,C 180,E1 -8490.293,E2 -8490.293} C_VEL
LIN {X 0,Y 453.018,Z 339.667,A -85,B 0,C 180,E1 -8491.834,E2 -8491.834} C_VEL
LIN {X 0,Y 453.274,Z 333.939,A -85,B 0,C 180,E1 -8493.147,E2 -8493.147} C_VEL
LIN {X 0,Y 453.618,Z 326.935,A -85,B 0,C 180,E1 -8494.437,E2 -8494.437} C_VEL
LIN {X 0,Y 454.054,Z 318.089,A -85,B 0,C 180,E1 -8495.754,E2 -8495.754} C_VEL
LIN {X 0,Y 454.491,Z 308.727,A -85,B 0,C 180,E1 -8496.885,E2 -8496.885} C_VEL
LIN {X 0,Y 454.977,Z 298.511,A -85,B 0,C 180,E1 -8497.88,E2 -8497.88} C_VEL
LIN {X 0,Y 455.464,Z 286.452,A -85,B 0,C 180,E1 -8498.818,E2 -8498.818} C_VEL
LIN {X 0,Y 455.922,Z 275.325,A -85,B 0,C 180,E1 -8499.492,E2 -8499.492} C_VEL
LIN {X 0,Y 456.193,Z 262.402,A -85,B 0,C 180,E1 -8500.077,E2 -8500.077} C_VEL
LIN {X 0,Y 456.495,Z 249.972,A -85,B 0,C 180,E1 -8500.46,E2 -8500.46} C_VEL
LIN {X 0,Y 457.122,Z 196.976,A -85,B 0,C 180,E1 -8501.383,E2 -8501.383} C_VEL
LIN {X 0,Y 457.513,Z 156.521,A -85,B 0,C 180,E1 -8502.084,E2 -8502.084} C_VEL
LIN {X 0,Y 454.483,Z 141.647,A -85,B 0,C 180,E1 -8502.462,E2 -8502.462} C_VEL
LIN {X 0,Y 454.318,Z 136.366,A -85,B 0,C 180,E1 -8503.607,E2 -8503.607} C_VEL
LIN {X 0,Y 453.554,Z 131.989,A -85,B 0,C 180,E1 -8504.601,E2 -8504.601} C_VEL
LIN {X 0,Y 453.472,Z 132.002,A -85,B 0,C 180,E1 -8505.75,E2 -8505.75} C_VEL
LIN {X 0,Y 452.777,Z 132.091,A -85,B 0,C 180,E1 -8506.491,E2 -8506.491} C_VEL
LIN {X 0,Y 449.903,Z 132.447,A -85,B 0,C 180,E1 -8507.695,E2 -8507.695} C_VEL
LIN {X 0,Y 447.506,Z 132.74,A -85,B 0,C 180,E1 -8508.666,E2 -8508.666} C_VEL
LIN {X 0,Y 446.502,Z 132.867,A -85,B 0,C 180,E1 -8509.416,E2 -8509.416} C_VEL
LIN {X 0,Y 446.433,Z 132.876,A -85,B 0,C 180,E1 -8509.67,E2 -8509.67} C_VEL
LIN {X 0,Y 446.407,Z 132.876,A -85,B 0,C 180,E1 -8512.121,E2 -8512.121} C_VEL
LIN {X 0,Y 446.423,Z 132.879,A -85,B 0,C 180,E1 -8515.476,E2 -8515.476} C_VEL
LIN {X 0,Y 446.414,Z 132.874,A -85,B 0,C 180,E1 -8518.699,E2 -8518.699} C_VEL
LIN {X 0,Y 446.484,Z 132.868,A -85,B 0,C 180,E1 -8521.821,E2 -8521.821} C_VEL
LIN {X 0,Y 446.456,Z 132.87,A -85,B 0,C 180,E1 -8524.847,E2 -8524.847} C_VEL
LIN {X 0,Y 446.447,Z 132.869,A -85,B 0,C 180,E1 -8528.245,E2 -8528.245} C_VEL
LIN {X 0,Y 446.451,Z 132.871,A -85,B 0,C 180,E1 -8531.649,E2 -8531.649} C_VEL
LIN {X 0,Y 446.507,Z 132.863,A -85,B 0,C 180,E1 -8534.479,E2 -8534.479} C_VEL
LIN {X 0,Y 446.517,Z 132.861,A -85,B 0,C 180,E1 -8538.193,E2 -8538.193} C_VEL
LIN {X 0,Y 446.599,Z 132.85,A -85,B 0,C 180,E1 -8541.857,E2 -8541.857} C_VEL
LIN {X 0,Y 446.64,Z 132.849,A -85,B 0,C 180,E1 -8544.582,E2 -8544.582} C_VEL
LIN {X 0,Y 446.708,Z 132.839,A -85,B 0,C 180,E1 -8547.294,E2 -8547.294} C_VEL
LIN {X 0,Y 446.793,Z 132.826,A -85,B 0,C 180,E1 -8550,E2 -8550} C_VEL
LIN {X 0,Y 446.707,Z 132.844,A -85,B 0,C 180,E1 -8552.705,E2 -8552.705} C_VEL
LIN {X 0,Y 446.638,Z 132.849,A -85,B 0,C 180,E1 -8556.323,E2 -8556.323} C_VEL
LIN {X 0,Y 446.536,Z 132.861,A -85,B 0,C 180,E1 -8559.055,E2 -8559.055} C_VEL
LIN {X 0,Y 446.519,Z 132.866,A -85,B 0,C 180,E1 -8562.729,E2 -8562.729} C_VEL
LIN {X 0,Y 446.494,Z 132.868,A -85,B 0,C 180,E1 -8566.228,E2 -8566.228} C_VEL
LIN {X 0,Y 446.467,Z 132.867,A -85,B 0,C 180,E1 -8569.303,E2 -8569.303} C_VEL
LIN {X 0,Y 446.416,Z 132.879,A -85,B 0,C 180,E1 -8572.199,E2 -8572.199} C_VEL
LIN {X 0,Y 446.441,Z 132.87,A -85,B 0,C 180,E1 -8575.153,E2 -8575.153} C_VEL
LIN {X 0,Y 446.481,Z 132.873,A -85,B 0,C 180,E1 -8578.178,E2 -8578.178} C_VEL
LIN {X 0,Y 446.417,Z 132.873,A -85,B 0,C 180,E1 -8581.3,E2 -8581.3} C_VEL
LIN {X 0,Y 446.427,Z 132.874,A -85,B 0,C 180,E1 -8584.523,E2 -8584.523} C_VEL
LIN {X 0,Y 446.427,Z 132.878,A -85,B 0,C 180,E1 -8588.082,E2 -8588.082} C_VEL
LIN {X 0,Y 446.427,Z 132.872,A -85,B 0,C 180,E1 -8590.918,E2 -8590.918} C_VEL
LIN {X 0,Y 446.442,Z 132.878,A -85,B 0,C 180,E1 -8593.84,E2 -8593.84} C_VEL
LIN {X 0,Y 446.396,Z 132.877,A -85,B 0,C 180,E1 -8596.403,E2 -8596.403} C_VEL
LIN {X 0,Y 446.464,Z 132.874,A -85,B 0,C 180,E1 -8599.805,E2 -8599.805} C_VEL
LIN {X 0,Y 446.428,Z 132.874,A -85,B 0,C 180,E1 -8602.124,E2 -8602.124} C_VEL
LIN {X 0,Y 446.426,Z 132.878,A -85,B 0,C 180,E1 -8605.477,E2 -8605.477} C_VEL
LIN {X 0,Y 446.413,Z 132.874,A -85,B 0,C 180,E1 -8608.7,E2 -8608.7} C_VEL
LIN {X 0,Y 446.481,Z 132.868,A -85,B 0,C 180,E1 -8611.822,E2 -8611.822} C_VEL
LIN {X 0,Y 446.454,Z 132.87,A -85,B 0,C 180,E1 -8614.848,E2 -8614.848} C_VEL
LIN {X 0,Y 446.445,Z 132.87,A -85,B 0,C 180,E1 -8618.245,E2 -8618.245} C_VEL
LIN {X 0,Y 446.455,Z 132.871,A -85,B 0,C 180,E1 -8621.649,E2 -8621.649} C_VEL
LIN {X 0,Y 446.505,Z 132.863,A -85,B 0,C 180,E1 -8624.48,E2 -8624.48} C_VEL
LIN {X 0,Y 446.515,Z 132.861,A -85,B 0,C 180,E1 -8628.193,E2 -8628.193} C_VEL
LIN {X 0,Y 446.598,Z 132.851,A -85,B 0,C 180,E1 -8631.858,E2 -8631.858} C_VEL
LIN {X 0,Y 446.64,Z 132.848,A -85,B 0,C 180,E1 -8634.583,E2 -8634.583} C_VEL
LIN {X 0,Y 446.707,Z 132.84,A -85,B 0,C 180,E1 -8637.295,E2 -8637.295} C_VEL
LIN {X 0,Y 446.792,Z 132.826,A -85,B 0,C 180,E1 -8640,E2 -8640} C_VEL
LIN {X 0,Y 446.707,Z 132.843,A -85,B 0,C 180,E1 -8642.706,E2 -8642.706} C_VEL
LIN {X 0,Y 446.646,Z 132.847,A -85,B 0,C 180,E1 -8646.324,E2 -8646.324} C_VEL
LIN {X 0,Y 446.537,Z 132.861,A -85,B 0,C 180,E1 -8649.056,E2 -8649.056} C_VEL
LIN {X 0,Y 446.52,Z 132.866,A -85,B 0,C 180,E1 -8652.73,E2 -8652.73} C_VEL
LIN {X 0,Y 446.495,Z 132.867,A -85,B 0,C 180,E1 -8656.228,E2 -8656.228} C_VEL
LIN {X 0,Y 446.468,Z 132.867,A -85,B 0,C 180,E1 -8659.304,E2 -8659.304} C_VEL
LIN {X 0,Y 446.417,Z 132.878,A -85,B 0,C 180,E1 -8662.2,E2 -8662.2} C_VEL
LIN {X 0,Y 446.443,Z 132.87,A -85,B 0,C 180,E1 -8665.154,E2 -8665.154} C_VEL
LIN {X 0,Y 446.484,Z 132.871,A -85,B 0,C 180,E1 -8668.179,E2 -8668.179} C_VEL
LIN {X 0,Y 446.418,Z 132.876,A -85,B 0,C 180,E1 -8671.775,E2 -8671.775} C_VEL
LIN {X 0,Y 446.428,Z 132.875,A -85,B 0,C 180,E1 -8674.523,E2 -8674.523} C_VEL
LIN {X 0,Y 446.435,Z 132.878,A -85,B 0,C 180,E1 -8678.083,E2 -8678.083} C_VEL
LIN {X 0,Y 446.443,Z 132.87,A -85,B 0,C 180,E1 -8680.921,E2 -8680.921} C_VEL
LIN {X 0,Y 446.417,Z 132.88,A -85,B 0,C 180,E1 -8683.844,E2 -8683.844} C_VEL
LIN {X 0,Y 446.399,Z 132.877,A -85,B 0,C 180,E1 -8686.404,E2 -8686.404} C_VEL
LIN {X 0,Y 446.427,Z 132.872,A -85,B 0,C 180,E1 -8689.083,E2 -8689.083} C_VEL
LIN {X 0,Y 446.41,Z 132.877,A -85,B 0,C 180,E1 -8692.122,E2 -8692.122} C_VEL
LIN {X 0,Y 446.43,Z 132.876,A -85,B 0,C 180,E1 -8695.478,E2 -8695.478} C_VEL
LIN {X 0,Y 446.417,Z 132.875,A -85,B 0,C 180,E1 -8698.7,E2 -8698.7} C_VEL
LIN {X 0,Y 446.518,Z 132.865,A -85,B 0,C 180,E1 -8702.334,E2 -8702.334} C_VEL
LIN {X 0,Y 446.574,Z 133.185,A -85,B 0,C 180,E1 -8702.465,E2 -8702.465} C_VEL
LIN {X 0,Y 449.212,Z 146.647,A -85,B 0,C 180,E1 -8705.013,E2 -8705.013} C_VEL
LIN {X 0,Y 448.574,Z 161.358,A -85,B 0,C 180,E1 -8707.575,E2 -8707.575} C_VEL
LIN {X 0,Y 447.679,Z 181.242,A -85,B 0,C 180,E1 -8710.989,E2 -8710.989} C_VEL
LIN {X 0,Y 447.276,Z 188.704,A -85,B 0,C 180,E1 -8712.258,E2 -8712.258} C_VEL
LIN {X 0,Y 450.445,Z 211.72,A -85,B 0,C 180,E1 -8712.804,E2 -8712.804} C_VEL
LIN {X 0,Y 449.45,Z 297.735,A -85,B 0,C 180,E1 -8714.323,E2 -8714.323} C_VEL
LIN {X 0,Y 448.97,Z 311.389,A -85,B 0,C 180,E1 -8714.742,E2 -8714.742} C_VEL
LIN {X 0,Y 448.488,Z 323.831,A -85,B 0,C 180,E1 -8715.306,E2 -8715.306} C_VEL
LIN {X 0,Y 447.87,Z 335.788,A -85,B 0,C 180,E1 -8716.039,E2 -8716.039} C_VEL
LIN {X 0,Y 447.327,Z 348.025,A -85,B 0,C 180,E1 -8717.011,E2 -8717.011} C_VEL
LIN {X 0,Y 446.902,Z 357.717,A -85,B 0,C 180,E1 -8717.974,E2 -8717.974} C_VEL
LIN {X 0,Y 446.4,Z 367.049,A -85,B 0,C 180,E1 -8719.11,E2 -8719.11} C_VEL
LIN {X 0,Y 445.976,Z 376.127,A -85,B 0,C 180,E1 -8720.476,E2 -8720.476} C_VEL
LIN {X 0,Y 445.72,Z 383.425,A -85,B 0,C 180,E1 -8721.842,E2 -8721.842} C_VEL
LIN {X 0,Y 445.535,Z 389.221,A -85,B 0,C 180,E1 -8723.206,E2 -8723.206} C_VEL
LIN {X 0,Y 445.486,Z 393.771,A -85,B 0,C 180,E1 -8724.569,E2 -8724.569} C_VEL
LIN {X 0,Y 445.421,Z 396.158,A -85,B 0,C 180,E1 -8725.475,E2 -8725.475} C_VEL
LIN {X 0,Y 445.452,Z 398.107,A -85,B 0,C 180,E1 -8726.382,E2 -8726.382} C_VEL
LIN {X 0,Y 445.478,Z 399.605,A -85,B 0,C 180,E1 -8727.288,E2 -8727.288} C_VEL
LIN {X 0,Y 445.454,Z 400.64,A -85,B 0,C 180,E1 -8728.192,E2 -8728.192} C_VEL
LIN {X 0,Y 445.438,Z 401.271,A -85,B 0,C 180,E1 -8729.096,E2 -8729.096} C_VEL
LIN {X 0,Y 445.418,Z 401.501,A -85,B 0,C 180,E1 -8730,E2 -8730} C_VEL
LIN {X 0,Y 445.437,Z 401.297,A -85,B 0,C 180,E1 -8730.904,E2 -8730.904} C_VEL
LIN {X 0,Y 445.429,Z 400.66,A -85,B 0,C 180,E1 -8731.809,E2 -8731.809} C_VEL
LIN {X 0,Y 445.476,Z 399.625,A -85,B 0,C 180,E1 -8732.713,E2 -8732.713} C_VEL
LIN {X 0,Y 445.436,Z 398.173,A -85,B 0,C 180,E1 -8733.619,E2 -8733.619} C_VEL
LIN {X 0,Y 445.481,Z 395.128,A -85,B 0,C 180,E1 -8734.978,E2 -8734.978} C_VEL
LIN {X 0,Y 445.456,Z 391.008,A -85,B 0,C 180,E1 -8736.341,E2 -8736.341} C_VEL
LIN {X 0,Y 445.69,Z 384.688,A -85,B 0,C 180,E1 -8737.931,E2 -8737.931} C_VEL
LIN {X 0,Y 445.916,Z 377.791,A -85,B 0,C 180,E1 -8739.297,E2 -8739.297} C_VEL
LIN {X 0,Y 446.299,Z 369.254,A -85,B 0,C 180,E1 -8740.663,E2 -8740.663} C_VEL
LIN {X 0,Y 446.819,Z 360.484,A -85,B 0,C 180,E1 -8741.799,E2 -8741.799} C_VEL
LIN {X 0,Y 447.258,Z 350.412,A -85,B 0,C 180,E1 -8742.87,E2 -8742.87} C_VEL
LIN {X 0,Y 447.926,Z 339.019,A -85,B 0,C 180,E1 -8743.844,E2 -8743.844} C_VEL
LIN {X 0,Y 448.553,Z 327.251,A -85,B 0,C 180,E1 -8744.635,E2 -8744.635} C_VEL
LIN {X 0,Y 449.212,Z 313.857,A -85,B 0,C 180,E1 -8745.309,E2 -8745.309} C_VEL
LIN {X 0,Y 449.704,Z 301.257,A -85,B 0,C 180,E1 -8745.756,E2 -8745.756} C_VEL
LIN {X 0,Y 449.996,Z 285.344,A -85,B 0,C 180,E1 -8746.095,E2 -8746.095} C_VEL
LIN {X 0,Y 450.843,Z 211.059,A -85,B 0,C 180,E1 -8747.429,E2 -8747.429} C_VEL
LIN {X 0,Y 447.987,Z 190.5,A -85,B 0,C 180,E1 -8747.952,E2 -8747.952} C_VEL
LIN {X 0,Y 447.338,Z 186.537,A -85,B 0,C 180,E1 -8748.09,E2 -8748.09} C_VEL
LIN {X 0,Y 447.877,Z 172.61,A -85,B 0,C 180,E1 -8750.435,E2 -8750.435} C_VEL
LIN {X 0,Y 448.579,Z 158.35,A -85,B 0,C 180,E1 -8752.855,E2 -8752.855} C_VEL
LIN {X 0,Y 449.14,Z 145.928,A -85,B 0,C 180,E1 -8754.992,E2 -8754.992} C_VEL
LIN {X 0,Y 446.921,Z 134.671,A -85,B 0,C 180,E1 -8757.132,E2 -8757.132} C_VEL
LIN {X 0,Y 446.516,Z 132.87,A -85,B 0,C 180,E1 -8757.507,E2 -8757.507} C_VEL
LIN {X 0,Y 446.431,Z 132.883,A -85,B 0,C 180,E1 -8760.25,E2 -8760.25} C_VEL
LIN {X 0,Y 446.449,Z 132.873,A -85,B 0,C 180,E1 -8763.454,E2 -8763.454} C_VEL
LIN {X 0,Y 446.405,Z 132.878,A -85,B 0,C 180,E1 -8766.745,E2 -8766.745} C_VEL
LIN {X 0,Y 446.482,Z 132.87,A -85,B 0,C 180,E1 -8769.529,E2 -8769.529} C_VEL
LIN {X 0,Y 446.433,Z 132.875,A -85,B 0,C 180,E1 -8772.605,E2 -8772.605} C_VEL
LIN {X 0,Y 446.457,Z 132.87,A -85,B 0,C 180,E1 -8775.103,E2 -8775.103} C_VEL
LIN {X 0,Y 446.431,Z 132.87,A -85,B 0,C 180,E1 -8778.609,E2 -8778.609} C_VEL
LIN {X 0,Y 446.441,Z 132.868,A -85,B 0,C 180,E1 -8780.972,E2 -8780.972} C_VEL
LIN {X 0,Y 446.421,Z 132.872,A -85,B 0,C 180,E1 -8784.374,E2 -8784.374} C_VEL
LIN {X 0,Y 446.423,Z 132.876,A -85,B 0,C 180,E1 -8787.638,E2 -8787.638} C_VEL
LIN {X 0,Y 446.451,Z 132.871,A -85,B 0,C 180,E1 -8790.79,E2 -8790.79} C_VEL
LIN {X 0,Y 446.481,Z 132.865,A -85,B 0,C 180,E1 -8793.848,E2 -8793.848} C_VEL
LIN {X 0,Y 446.432,Z 132.875,A -85,B 0,C 180,E1 -8796.823,E2 -8796.823} C_VEL
LIN {X 0,Y 446.447,Z 132.871,A -85,B 0,C 180,E1 -8799.737,E2 -8799.737} C_VEL
LIN {X 0,Y 446.458,Z 132.869,A -85,B 0,C 180,E1 -8802.597,E2 -8802.597} C_VEL
LIN {X 0,Y 446.471,Z 132.87,A -85,B 0,C 180,E1 -8805.412,E2 -8805.412} C_VEL
LIN {X 0,Y 446.52,Z 132.864,A -85,B 0,C 180,E1 -8808.193,E2 -8808.193} C_VEL
LIN {X 0,Y 446.535,Z 132.865,A -85,B 0,C 180,E1 -8810.944,E2 -8810.944} C_VEL
LIN {X 0,Y 446.624,Z 132.852,A -85,B 0,C 180,E1 -8813.676,E2 -8813.676} C_VEL
LIN {X 0,Y 446.685,Z 132.846,A -85,B 0,C 180,E1 -8817.294,E2 -8817.294} C_VEL
LIN {X 0,Y 446.791,Z 132.832,A -85,B 0,C 180,E1 -8820,E2 -8820} C_VEL
LIN {X 0,Y 446.679,Z 132.848,A -85,B 0,C 180,E1 -8822.705,E2 -8822.705} C_VEL
LIN {X 0,Y 446.531,Z 132.963,A -85,B 0,C 180,E1 -8824.739,E2 -8824.739} C_VEL
LIN {X 0,Y 448.121,Z 141.068,A -85,B 0,C 180,E1 -8826.529,E2 -8826.529} C_VEL
LIN {X 0,Y 448.14,Z 143.516,A -85,B 0,C 180,E1 -8827.037,E2 -8827.037} C_VEL
LIN {X 0,Y 451.474,Z 158.188,A -85,B 0,C 180,E1 -8827.491,E2 -8827.491} C_VEL
LIN {X 0,Y 450.134,Z 251.536,A -85,B 0,C 180,E1 -8829.204,E2 -8829.204} C_VEL
LIN {X 0,Y 449.829,Z 265.346,A -85,B 0,C 180,E1 -8829.655,E2 -8829.655} C_VEL
LIN {X 0,Y 449.465,Z 277.624,A -85,B 0,C 180,E1 -8830.245,E2 -8830.245} C_VEL
LIN {X 0,Y 448.866,Z 290.255,A -85,B 0,C 180,E1 -8831.058,E2 -8831.058} C_VEL
LIN {X 0,Y 448.345,Z 301.445,A -85,B 0,C 180,E1 -8831.987,E2 -8831.987} C_VEL
LIN {X 0,Y 447.732,Z 312.182,A -85,B 0,C 180,E1 -8833.114,E2 -8833.114} C_VEL
LIN {X 0,Y 447.2,Z 321.539,A -85,B 0,C 180,E1 -8834.33,E2 -8834.33} C_VEL
LIN {X 0,Y 446.775,Z 328.939,A -85,B 0,C 180,E1 -8835.51,E2 -8835.51} C_VEL
LIN {X 0,Y 446.34,Z 336.138,A -85,B 0,C 180,E1 -8836.935,E2 -8836.935} C_VEL
LIN {X 0,Y 446.033,Z 341.852,A -85,B 0,C 180,E1 -8838.369,E2 -8838.369} C_VEL
LIN {X 0,Y 445.795,Z 346.282,A -85,B 0,C 180,E1 -8839.812,E2 -8839.812} C_VEL
LIN {X 0,Y 445.586,Z 349.908,A -85,B 0,C 180,E1 -8841.474,E2 -8841.474} C_VEL
LIN {X 0,Y 445.412,Z 352.124,A -85,B 0,C 180,E1 -8843.232,E2 -8843.232} C_VEL
LIN {X 0,Y 445.352,Z 352.721,A -85,B 0,C 180,E1 -8844.223,E2 -8844.223} C_VEL
LIN {X 0,Y 445.398,Z 352.54,A -85,B 0,C 180,E1 -8845.919,E2 -8845.919} C_VEL
LIN {X 0,Y 445.402,Z 351.447,A -85,B 0,C 180,E1 -8847.231,E2 -8847.231} C_VEL
LIN {X 0,Y 445.465,Z 349.977,A -85,B 0,C 180,E1 -8848.249,E2 -8848.249} C_VEL
LIN {X 0,Y 445.688,Z 346.581,A -85,B 0,C 180,E1 -8849.855,E2 -8849.855} C_VEL
LIN {X 0,Y 445.833,Z 342.101,A -85,B 0,C 180,E1 -8851.345,E2 -8851.345} C_VEL
LIN {X 0,Y 446.18,Z 335.876,A -85,B 0,C 180,E1 -8852.902,E2 -8852.902} C_VEL
LIN {X 0,Y 446.471,Z 329.084,A -85,B 0,C 180,E1 -8854.246,E2 -8854.246} C_VEL
LIN {X 0,Y 446.956,Z 320.716,A -85,B 0,C 180,E1 -8855.576,E2 -8855.576} C_VEL
LIN {X 0,Y 447.389,Z 311.509,A -85,B 0,C 180,E1 -8856.759,E2 -8856.759} C_VEL
LIN {X 0,Y 447.914,Z 301.09,A -85,B 0,C 180,E1 -8857.845,E2 -8857.845} C_VEL
LIN {X 0,Y 448.417,Z 290.36,A -85,B 0,C 180,E1 -8858.744,E2 -8858.744} C_VEL
LIN {X 0,Y 448.86,Z 278.914,A -85,B 0,C 180,E1 -8859.5,E2 -8859.5} C_VEL
LIN {X 0,Y 449.266,Z 265.763,A -85,B 0,C 180,E1 -8860.157,E2 -8860.157} C_VEL
LIN {X 0,Y 449.512,Z 253.073,A -85,B 0,C 180,E1 -8860.597,E2 -8860.597} C_VEL
LIN {X 0,Y 449.749,Z 236.329,A -85,B 0,C 180,E1 -8860.937,E2 -8860.937} C_VEL
LIN {X 0,Y 450.682,Z 157.504,A -85,B 0,C 180,E1 -8862.315,E2 -8862.315} C_VEL
LIN {X 0,Y 447.54,Z 141.967,A -85,B 0,C 180,E1 -8862.716,E2 -8862.716} C_VEL
LIN {X 0,Y 447.295,Z 137.328,A -85,B 0,C 180,E1 -8863.736,E2 -8863.736} C_VEL
LIN {X 0,Y 446.493,Z 132.869,A -85,B 0,C 180,E1 -8864.781,E2 -8864.781} C_VEL
LIN {X 0,Y 446.428,Z 132.872,A -85,B 0,C 180,E1 -8868.609,E2 -8868.609} C_VEL
LIN {X 0,Y 446.433,Z 132.876,A -85,B 0,C 180,E1 -8869.67,E2 -8869.67} C_VEL
LIN {X 0,Y 445.786,Z 132.961,A -85,B 0,C 180,E1 -8870.423,E2 -8870.423} C_VEL
LIN {X 0,Y 442.895,Z 133.32,A -85,B 0,C 180,E1 -8871.644,E2 -8871.644} C_VEL
LIN {X 0,Y 440.453,Z 133.619,A -85,B 0,C 180,E1 -8872.63,E2 -8872.63} C_VEL
LIN {X 0,Y 439.433,Z 133.748,A -85,B 0,C 180,E1 -8873.393,E2 -8873.393} C_VEL
LIN {X 0,Y 439.368,Z 133.757,A -85,B 0,C 180,E1 -8873.651,E2 -8873.651} C_VEL
LIN {X 0,Y 439.395,Z 133.748,A -85,B 0,C 180,E1 -8876.276,E2 -8876.276} C_VEL
LIN {X 0,Y 439.38,Z 133.754,A -85,B 0,C 180,E1 -8879.739,E2 -8879.739} C_VEL
LIN {X 0,Y 439.441,Z 133.742,A -85,B 0,C 180,E1 -8882.367,E2 -8882.367} C_VEL
LIN {X 0,Y 439.414,Z 133.748,A -85,B 0,C 180,E1 -8885.735,E2 -8885.735} C_VEL
LIN {X 0,Y 439.388,Z 133.755,A -85,B 0,C 180,E1 -8889.397,E2 -8889.397} C_VEL
LIN {X 0,Y 439.404,Z 133.747,A -85,B 0,C 180,E1 -8892.308,E2 -8892.308} C_VEL
LIN {X 0,Y 439.447,Z 133.749,A -85,B 0,C 180,E1 -8895.174,E2 -8895.174} C_VEL
LIN {X 0,Y 439.483,Z 133.737,A -85,B 0,C 180,E1 -8898.001,E2 -8898.001} C_VEL
LIN {X 0,Y 439.547,Z 133.729,A -85,B 0,C 180,E1 -8901.726,E2 -8901.726} C_VEL
LIN {X 0,Y 439.616,Z 133.723,A -85,B 0,C 180,E1 -8904.495,E2 -8904.495} C_VEL
LIN {X 0,Y 439.635,Z 133.719,A -85,B 0,C 180,E1 -8908.167,E2 -8908.167} C_VEL
LIN {X 0,Y 439.763,Z 133.702,A -85,B 0,C 180,E1 -8910,E2 -8910} C_VEL
LIN {X 0,Y 439.653,Z 133.723,A -85,B 0,C 180,E1 -8912.748,E2 -8912.748} C_VEL
LIN {X 0,Y 439.61,Z 133.725,A -85,B 0,C 180,E1 -8916.425,E2 -8916.425} C_VEL
LIN {X 0,Y 439.498,Z 133.736,A -85,B 0,C 180,E1 -8919.201,E2 -8919.201} C_VEL
LIN {X 0,Y 439.463,Z 133.742,A -85,B 0,C 180,E1 -8922.937,E2 -8922.937} C_VEL
LIN {X 0,Y 439.445,Z 133.748,A -85,B 0,C 180,E1 -8926.349,E2 -8926.349} C_VEL
LIN {X 0,Y 439.4,Z 133.748,A -85,B 0,C 180,E1 -8929.626,E2 -8929.626} C_VEL
LIN {X 0,Y 439.361,Z 133.756,A -85,B 0,C 180,E1 -8932.575,E2 -8932.575} C_VEL
LIN {X 0,Y 439.394,Z 133.749,A -85,B 0,C 180,E1 -8935.585,E2 -8935.585} C_VEL
LIN {X 0,Y 439.422,Z 133.747,A -85,B 0,C 180,E1 -8938.673,E2 -8938.673} C_VEL
LIN {X 0,Y 439.38,Z 133.756,A -85,B 0,C 180,E1 -8942.033,E2 -8942.033} C_VEL
LIN {X 0,Y 439.393,Z 133.749,A -85,B 0,C 180,E1 -8945.341,E2 -8945.341} C_VEL
LIN {X 0,Y 439.385,Z 133.75,A -85,B 0,C 180,E1 -8948.594,E2 -8948.594} C_VEL
LIN {X 0,Y 439.391,Z 133.749,A -85,B 0,C 180,E1 -8951.258,E2 -8951.258} C_VEL
LIN {X 0,Y 439.405,Z 133.747,A -85,B 0,C 180,E1 -8954.728,E2 -8954.728} C_VEL
LIN {X 0,Y 439.394,Z 133.756,A -85,B 0,C 180,E1 -8957.796,E2 -8957.796} C_VEL
LIN {X 0,Y 439.446,Z 133.743,A -85,B 0,C 180,E1 -8960.23,E2 -8960.23} C_VEL
LIN {X 0,Y 439.372,Z 133.758,A -85,B 0,C 180,E1 -8963.713,E2 -8963.713} C_VEL
LIN {X 0,Y 439.369,Z 133.753,A -85,B 0,C 180,E1 -8967.054,E2 -8967.054} C_VEL
LIN {X 0,Y 439.379,Z 133.75,A -85,B 0,C 180,E1 -8970.274,E2 -8970.274} C_VEL
LIN {X 0,Y 439.425,Z 133.751,A -85,B 0,C 180,E1 -8973.396,E2 -8973.396} C_VEL
LIN {X 0,Y 439.383,Z 133.749,A -85,B 0,C 180,E1 -8976.43,E2 -8976.43} C_VEL
LIN {X 0,Y 439.387,Z 133.756,A -85,B 0,C 180,E1 -8979.397,E2 -8979.397} C_VEL
LIN {X 0,Y 439.429,Z 133.744,A -85,B 0,C 180,E1 -8982.31,E2 -8982.31} C_VEL
LIN {X 0,Y 439.445,Z 133.749,A -85,B 0,C 180,E1 -8985.174,E2 -8985.174} C_VEL
LIN {X 0,Y 439.481,Z 133.737,A -85,B 0,C 180,E1 -8988.002,E2 -8988.002} C_VEL
LIN {X 0,Y 439.546,Z 133.73,A -85,B 0,C 180,E1 -8991.727,E2 -8991.727} C_VEL
LIN {X 0,Y 439.615,Z 133.722,A -85,B 0,C 180,E1 -8994.496,E2 -8994.496} C_VEL
LIN {X 0,Y 439.634,Z 133.718,A -85,B 0,C 180,E1 -8998.168,E2 -8998.168} C_VEL
LIN {X 0,Y 439.762,Z 133.702,A -85,B 0,C 180,E1 -9000,E2 -9000} C_VEL
LIN {X 0,Y 439.653,Z 133.723,A -85,B 0,C 180,E1 -9002.749,E2 -9002.749} C_VEL
LIN {X 0,Y 439.618,Z 133.724,A -85,B 0,C 180,E1 -9006.426,E2 -9006.426} C_VEL
LIN {X 0,Y 439.499,Z 133.737,A -85,B 0,C 180,E1 -9009.202,E2 -9009.202} C_VEL
LIN {X 0,Y 439.464,Z 133.743,A -85,B 0,C 180,E1 -9012.938,E2 -9012.938} C_VEL
LIN {X 0,Y 439.446,Z 133.747,A -85,B 0,C 180,E1 -9016.349,E2 -9016.349} C_VEL
LIN {X 0,Y 439.402,Z 133.747,A -85,B 0,C 180,E1 -9019.627,E2 -9019.627} C_VEL
LIN {X 0,Y 439.363,Z 133.757,A -85,B 0,C 180,E1 -9022.576,E2 -9022.576} C_VEL
LIN {X 0,Y 439.396,Z 133.748,A -85,B 0,C 180,E1 -9025.586,E2 -9025.586} C_VEL
LIN {X 0,Y 439.416,Z 133.748,A -85,B 0,C 180,E1 -9028.674,E2 -9028.674} C_VEL
LIN {X 0,Y 439.369,Z 133.757,A -85,B 0,C 180,E1 -9032.031,E2 -9032.031} C_VEL
LIN {X 0,Y 439.394,Z 133.748,A -85,B 0,C 180,E1 -9035.341,E2 -9035.341} C_VEL
LIN {X 0,Y 439.395,Z 133.749,A -85,B 0,C 180,E1 -9038.594,E2 -9038.594} C_VEL
LIN {X 0,Y 439.398,Z 133.748,A -85,B 0,C 180,E1 -9041.259,E2 -9041.259} C_VEL
LIN {X 0,Y 439.403,Z 133.747,A -85,B 0,C 180,E1 -9044.729,E2 -9044.729} C_VEL
LIN {X 0,Y 439.396,Z 133.755,A -85,B 0,C 180,E1 -9047.796,E2 -9047.796} C_VEL
LIN {X 0,Y 439.426,Z 133.746,A -85,B 0,C 180,E1 -9050.228,E2 -9050.228} C_VEL
LIN {X 0,Y 439.374,Z 133.758,A -85,B 0,C 180,E1 -9053.713,E2 -9053.713} C_VEL
LIN {X 0,Y 439.373,Z 133.752,A -85,B 0,C 180,E1 -9057.055,E2 -9057.055} C_VEL
LIN {X 0,Y 439.383,Z 133.751,A -85,B 0,C 180,E1 -9060.275,E2 -9060.275} C_VEL
LIN {X 0,Y 439.464,Z 133.752,A -85,B 0,C 180,E1 -9062.192,E2 -9062.192} C_VEL
LIN {X 0,Y 441.936,Z 146.098,A -85,B 0,C 180,E1 -9064.573,E2 -9064.573} C_VEL
LIN {X 0,Y 442.306,Z 149.847,A -85,B 0,C 180,E1 -9065.267,E2 -9065.267} C_VEL
LIN {X 0,Y 441.242,Z 168.3,A -85,B 0,C 180,E1 -9068.51,E2 -9068.51} C_VEL
LIN {X 0,Y 440.462,Z 184.861,A -85,B 0,C 180,E1 -9071.391,E2 -9071.391} C_VEL
LIN {X 0,Y 440.262,Z 188.567,A -85,B 0,C 180,E1 -9072.02,E2 -9072.02} C_VEL
LIN {X 0,Y 443.555,Z 213.034,A -85,B 0,C 180,E1 -9072.591,E2 -9072.591} C_VEL
LIN {X 0,Y 442.532,Z 298.192,A -85,B 0,C 180,E1 -9074.13,E2 -9074.13} C_VEL
LIN {X 0,Y 442.019,Z 311.559,A -85,B 0,C 180,E1 -9074.555,E2 -9074.555} C_VEL
LIN {X 0,Y 441.543,Z 323.843,A -85,B 0,C 180,E1 -9075.128,E2 -9075.128} C_VEL
LIN {X 0,Y 440.845,Z 336.493,A -85,B 0,C 180,E1 -9075.93,E2 -9075.93} C_VEL
LIN {X 0,Y 440.293,Z 347.545,A -85,B 0,C 180,E1 -9076.828,E2 -9076.828} C_VEL
LIN {X 0,Y 439.856,Z 358.031,A -85,B 0,C 180,E1 -9077.895,E2 -9077.895} C_VEL
LIN {X 0,Y 439.283,Z 368.069,A -85,B 0,C 180,E1 -9079.165,E2 -9079.165} C_VEL
LIN {X 0,Y 438.861,Z 376.9,A -85,B 0,C 180,E1 -9080.553,E2 -9080.553} C_VEL
LIN {X 0,Y 438.606,Z 383.93,A -85,B 0,C 180,E1 -9081.941,E2 -9081.941} C_VEL
LIN {X 0,Y 438.423,Z 390.372,A -85,B 0,C 180,E1 -9083.558,E2 -9083.558} C_VEL
LIN {X 0,Y 438.41,Z 394.57,A -85,B 0,C 180,E1 -9084.942,E2 -9084.942} C_VEL
LIN {X 0,Y 438.352,Z 397.664,A -85,B 0,C 180,E1 -9086.323,E2 -9086.323} C_VEL
LIN {X 0,Y 438.403,Z 399.183,A -85,B 0,C 180,E1 -9087.244,E2 -9087.244} C_VEL
LIN {X 0,Y 438.37,Z 400.228,A -85,B 0,C 180,E1 -9088.163,E2 -9088.163} C_VEL
LIN {X 0,Y 438.376,Z 400.869,A -85,B 0,C 180,E1 -9089.082,E2 -9089.082} C_VEL
LIN {X 0,Y 438.355,Z 401.105,A -85,B 0,C 180,E1 -9090,E2 -9090} C_VEL
LIN {X 0,Y 438.345,Z 400.914,A -85,B 0,C 180,E1 -9090.919,E2 -9090.919} C_VEL
LIN {X 0,Y 438.347,Z 400.283,A -85,B 0,C 180,E1 -9091.838,E2 -9091.838} C_VEL
LIN {X 0,Y 438.401,Z 399.25,A -85,B 0,C 180,E1 -9092.757,E2 -9092.757} C_VEL
LIN {X 0,Y 438.336,Z 397.802,A -85,B 0,C 180,E1 -9093.677,E2 -9093.677} C_VEL
LIN {X 0,Y 438.409,Z 394.766,A -85,B 0,C 180,E1 -9095.059,E2 -9095.059} C_VEL
LIN {X 0,Y 438.37,Z 390.655,A -85,B 0,C 180,E1 -9096.444,E2 -9096.444} C_VEL
LIN {X 0,Y 438.62,Z 384.354,A -85,B 0,C 180,E1 -9098.06,E2 -9098.06} C_VEL
LIN {X 0,Y 438.857,Z 377.466,A -85,B 0,C 180,E1 -9099.448,E2 -9099.448} C_VEL
LIN {X 0,Y 439.291,Z 368.938,A -85,B 0,C 180,E1 -9100.835,E2 -9100.835} C_VEL
LIN {X 0,Y 439.829,Z 360.201,A -85,B 0,C 180,E1 -9101.989,E2 -9101.989} C_VEL
LIN {X 0,Y 440.302,Z 350.166,A -85,B 0,C 180,E1 -9103.076,E2 -9103.076} C_VEL
LIN {X 0,Y 441.023,Z 338.821,A -85,B 0,C 180,E1 -9104.065,E2 -9104.065} C_VEL
LIN {X 0,Y 441.667,Z 327.147,A -85,B 0,C 180,E1 -9104.868,E2 -9104.868} C_VEL
LIN {X 0,Y 442.361,Z 313.855,A -85,B 0,C 180,E1 -9105.552,E2 -9105.552} C_VEL
LIN {X 0,Y 442.929,Z 300.539,A -85,B 0,C 180,E1 -9106.033,E2 -9106.033} C_VEL
LIN {X 0,Y 443.22,Z 284.617,A -85,B 0,C 180,E1 -9106.377,E2 -9106.377} C_VEL
LIN {X 0,Y 444.166,Z 212.028,A -85,B 0,C 180,E1 -9107.711,E2 -9107.711} C_VEL
LIN {X 0,Y 441.49,Z 192.468,A -85,B 0,C 180,E1 -9108.224,E2 -9108.224} C_VEL
LIN {X 0,Y 440.438,Z 186.137,A -85,B 0,C 180,E1 -9108.421,E2 -9108.421} C_VEL
LIN {X 0,Y 441.259,Z 168.212,A -85,B 0,C 180,E1 -9111.489,E2 -9111.489} C_VEL
LIN {X 0,Y 442.275,Z 149.529,A -85,B 0,C 180,E1 -9114.741,E2 -9114.741} C_VEL
LIN {X 0,Y 442.006,Z 145.808,A -85,B 0,C 180,E1 -9115.424,E2 -9115.424} C_VEL
LIN {X 0,Y 439.479,Z 133.765,A -85,B 0,C 180,E1 -9117.778,E2 -9117.778} C_VEL
LIN {X 0,Y 439.365,Z 133.761,A -85,B 0,C 180,E1 -9120.789,E2 -9120.789} C_VEL
LIN {X 0,Y 439.391,Z 133.755,A -85,B 0,C 180,E1 -9124.044,E2 -9124.044} C_VEL
LIN {X 0,Y 439.352,Z 133.756,A -85,B 0,C 180,E1 -9126.887,E2 -9126.887} C_VEL
LIN {X 0,Y 439.417,Z 133.752,A -85,B 0,C 180,E1 -9129.851,E2 -9129.851} C_VEL
LIN {X 0,Y 439.386,Z 133.753,A -85,B 0,C 180,E1 -9132.627,E2 -9132.627} C_VEL
LIN {X 0,Y 439.405,Z 133.75,A -85,B 0,C 180,E1 -9135.271,E2 -9135.271} C_VEL
LIN {X 0,Y 439.392,Z 133.746,A -85,B 0,C 180,E1 -9138.743,E2 -9138.743} C_VEL
LIN {X 0,Y 439.375,Z 133.752,A -85,B 0,C 180,E1 -9141.608,E2 -9141.608} C_VEL
LIN {X 0,Y 439.399,Z 133.747,A -85,B 0,C 180,E1 -9144.844,E2 -9144.844} C_VEL
LIN {X 0,Y 439.375,Z 133.749,A -85,B 0,C 180,E1 -9148.139,E2 -9148.139} C_VEL
LIN {X 0,Y 439.436,Z 133.746,A -85,B 0,C 180,E1 -9151.598,E2 -9151.598} C_VEL
LIN {X 0,Y 439.404,Z 133.745,A -85,B 0,C 180,E1 -9154.415,E2 -9154.415} C_VEL
LIN {X 0,Y 439.368,Z 133.756,A -85,B 0,C 180,E1 -9157.424,E2 -9157.424} C_VEL
LIN {X 0,Y 439.444,Z 133.745,A -85,B 0,C 180,E1 -9160.663,E2 -9160.663} C_VEL
LIN {X 0,Y 439.465,Z 133.74,A -85,B 0,C 180,E1 -9164.224,E2 -9164.224} C_VEL
LIN {X 0,Y 439.486,Z 133.739,A -85,B 0,C 180,E1 -9168.001,E2 -9168.001} C_VEL
LIN {X 0,Y 439.506,Z 133.738,A -85,B 0,C 180,E1 -9171.725,E2 -9171.725} C_VEL
LIN {X 0,Y 439.613,Z 133.729,A -85,B 0,C 180,E1 -9174.495,E2 -9174.495} C_VEL
LIN {X 0,Y 439.636,Z 133.726,A -85,B 0,C 180,E1 -9178.167,E2 -9178.167} C_VEL
LIN {X 0,Y 439.761,Z 133.708,A -85,B 0,C 180,E1 -9180,E2 -9180} C_VEL
LIN {X 0,Y 439.629,Z 133.727,A -85,B 0,C 180,E1 -9182.749,E2 -9182.749} C_VEL
LIN {X 0,Y 439.43,Z 133.87,A -85,B 0,C 180,E1 -9184.443,E2 -9184.443} C_VEL
LIN {X 0,Y 441.116,Z 141.494,A -85,B 0,C 180,E1 -9186.173,E2 -9186.173} C_VEL
LIN {X 0,Y 441.282,Z 143.879,A -85,B 0,C 180,E1 -9186.688,E2 -9186.688} C_VEL
LIN {X 0,Y 444.879,Z 159.813,A -85,B 0,C 180,E1 -9187.203,E2 -9187.203} C_VEL
LIN {X 0,Y 443.391,Z 251.47,A -85,B 0,C 180,E1 -9188.919,E2 -9188.919} C_VEL
LIN {X 0,Y 443.116,Z 264.85,A -85,B 0,C 180,E1 -9189.356,E2 -9189.356} C_VEL
LIN {X 0,Y 442.69,Z 277.465,A -85,B 0,C 180,E1 -9189.957,E2 -9189.957} C_VEL
LIN {X 0,Y 442.083,Z 289.967,A -85,B 0,C 180,E1 -9190.765,E2 -9190.765} C_VEL
LIN {X 0,Y 441.486,Z 301.329,A -85,B 0,C 180,E1 -9191.71,E2 -9191.71} C_VEL
LIN {X 0,Y 440.946,Z 311.501,A -85,B 0,C 180,E1 -9192.776,E2 -9192.776} C_VEL
LIN {X 0,Y 440.277,Z 321.601,A -85,B 0,C 180,E1 -9194.089,E2 -9194.089} C_VEL
LIN {X 0,Y 439.832,Z 329.054,A -85,B 0,C 180,E1 -9195.286,E2 -9195.286} C_VEL
LIN {X 0,Y 439.356,Z 336.323,A -85,B 0,C 180,E1 -9196.734,E2 -9196.734} C_VEL
LIN {X 0,Y 439.023,Z 342.078,A -85,B 0,C 180,E1 -9198.189,E2 -9198.189} C_VEL
LIN {X 0,Y 438.758,Z 346.552,A -85,B 0,C 180,E1 -9199.656,E2 -9199.656} C_VEL
LIN {X 0,Y 438.594,Z 348.897,A -85,B 0,C 180,E1 -9200.642,E2 -9200.642} C_VEL
LIN {X 0,Y 438.474,Z 350.683,A -85,B 0,C 180,E1 -9201.632,E2 -9201.632} C_VEL
LIN {X 0,Y 438.359,Z 352.02,A -85,B 0,C 180,E1 -9202.63,E2 -9202.63} C_VEL
LIN {X 0,Y 438.306,Z 353,A -85,B 0,C 180,E1 -9203.94,E2 -9203.94} C_VEL
LIN {X 0,Y 438.31,Z 353.067,A -85,B 0,C 180,E1 -9205.653,E2 -9205.653} C_VEL
LIN {X 0,Y 438.3,Z 352.395,A -85,B 0,C 180,E1 -9206.677,E2 -9206.677} C_VEL
LIN {X 0,Y 438.374,Z 350.571,A -85,B 0,C 180,E1 -9208.144,E2 -9208.144} C_VEL
LIN {X 0,Y 438.598,Z 347.243,A -85,B 0,C 180,E1 -9209.784,E2 -9209.784} C_VEL
LIN {X 0,Y 438.756,Z 342.635,A -85,B 0,C 180,E1 -9211.371,E2 -9211.371} C_VEL
LIN {X 0,Y 439.137,Z 336.378,A -85,B 0,C 180,E1 -9212.965,E2 -9212.965} C_VEL
LIN {X 0,Y 439.429,Z 329.682,A -85,B 0,C 180,E1 -9214.316,E2 -9214.316} C_VEL
LIN {X 0,Y 439.874,Z 322.259,A -85,B 0,C 180,E1 -9215.535,E2 -9215.535} C_VEL
LIN {X 0,Y 440.336,Z 313.116,A -85,B 0,C 180,E1 -9216.764,E2 -9216.764} C_VEL
LIN {X 0,Y 440.856,Z 303,A -85,B 0,C 180,E1 -9217.861,E2 -9217.861} C_VEL
LIN {X 0,Y 441.404,Z 292.181,A -85,B 0,C 180,E1 -9218.809,E2 -9218.809} C_VEL
LIN {X 0,Y 441.871,Z 281.174,A -85,B 0,C 180,E1 -9219.579,E2 -9219.579} C_VEL
LIN {X 0,Y 442.289,Z 268.458,A -85,B 0,C 180,E1 -9220.253,E2 -9220.253} C_VEL
LIN {X 0,Y 442.576,Z 254.676,A -85,B 0,C 180,E1 -9220.772,E2 -9220.772} C_VEL
LIN {X 0,Y 442.865,Z 239.801,A -85,B 0,C 180,E1 -9221.097,E2 -9221.097} C_VEL
LIN {X 0,Y 443.802,Z 158.197,A -85,B 0,C 180,E1 -9222.553,E2 -9222.553} C_VEL
LIN {X 0,Y 440.571,Z 142.225,A -85,B 0,C 180,E1 -9222.988,E2 -9222.988} C_VEL
LIN {X 0,Y 440.121,Z 137.439,A -85,B 0,C 180,E1 -9224.063,E2 -9224.063} C_VEL
LIN {X 0,Y 439.459,Z 133.745,A -85,B 0,C 180,E1 -9224.931,E2 -9224.931} C_VEL
LIN {X 0,Y 439.388,Z 133.749,A -85,B 0,C 180,E1 -9228.743,E2 -9228.743} C_VEL
LIN {X 0,Y 439.371,Z 133.758,A -85,B 0,C 180,E1 -9231.608,E2 -9231.608} C_VEL
LIN {X 0,Y 439.368,Z 133.757,A -85,B 0,C 180,E1 -9233.651,E2 -9233.651} C_VEL
LIN {X 0,Y 438.741,Z 133.842,A -85,B 0,C 180,E1 -9234.416,E2 -9234.416} C_VEL
LIN {X 0,Y 435.879,Z 134.204,A -85,B 0,C 180,E1 -9235.66,E2 -9235.66} C_VEL
LIN {X 0,Y 433.439,Z 134.505,A -85,B 0,C 180,E1 -9236.664,E2 -9236.664} C_VEL
LIN {X 0,Y 432.401,Z 134.627,A -85,B 0,C 180,E1 -9237.44,E2 -9237.44} C_VEL
LIN {X 0,Y 432.323,Z 134.634,A -85,B 0,C 180,E1 -9237.702,E2 -9237.702} C_VEL
LIN {X 0,Y 432.342,Z 134.627,A -85,B 0,C 180,E1 -9240.812,E2 -9240.812} C_VEL
LIN {X 0,Y 432.363,Z 134.625,A -85,B 0,C 180,E1 -9243.967,E2 -9243.967} C_VEL
LIN {X 0,Y 432.318,Z 134.633,A -85,B 0,C 180,E1 -9247.035,E2 -9247.035} C_VEL
LIN {X 0,Y 432.385,Z 134.622,A -85,B 0,C 180,E1 -9250.515,E2 -9250.515} C_VEL
LIN {X 0,Y 432.429,Z 134.616,A -85,B 0,C 180,E1 -9253.961,E2 -9253.961} C_VEL
LIN {X 0,Y 432.458,Z 134.612,A -85,B 0,C 180,E1 -9257.803,E2 -9257.803} C_VEL
LIN {X 0,Y 432.491,Z 134.609,A -85,B 0,C 180,E1 -9261.59,E2 -9261.59} C_VEL
LIN {X 0,Y 432.592,Z 134.597,A -85,B 0,C 180,E1 -9264.406,E2 -9264.406} C_VEL
LIN {X 0,Y 432.605,Z 134.594,A -85,B 0,C 180,E1 -9268.138,E2 -9268.138} C_VEL
LIN {X 0,Y 432.732,Z 134.578,A -85,B 0,C 180,E1 -9270,E2 -9270} C_VEL
LIN {X 0,Y 432.603,Z 134.601,A -85,B 0,C 180,E1 -9272.793,E2 -9272.793} C_VEL
LIN {X 0,Y 432.563,Z 134.605,A -85,B 0,C 180,E1 -9276.53,E2 -9276.53} C_VEL
LIN {X 0,Y 432.441,Z 134.615,A -85,B 0,C 180,E1 -9279.353,E2 -9279.353} C_VEL
LIN {X 0,Y 432.429,Z 134.62,A -85,B 0,C 180,E1 -9282.803,E2 -9282.803} C_VEL
LIN {X 0,Y 432.41,Z 134.625,A -85,B 0,C 180,E1 -9286.479,E2 -9286.479} C_VEL
LIN {X 0,Y 432.337,Z 134.63,A -85,B 0,C 180,E1 -9289.96,E2 -9289.96} C_VEL
LIN {X 0,Y 432.315,Z 134.631,A -85,B 0,C 180,E1 -9292.964,E2 -9292.964} C_VEL
LIN {X 0,Y 432.358,Z 134.629,A -85,B 0,C 180,E1 -9296.032,E2 -9296.032} C_VEL
LIN {X 0,Y 432.349,Z 134.625,A -85,B 0,C 180,E1 -9299.187,E2 -9299.187} C_VEL
LIN {X 0,Y 432.329,Z 134.633,A -85,B 0,C 180,E1 -9302.294,E2 -9302.294} C_VEL
LIN {X 0,Y 432.338,Z 134.628,A -85,B 0,C 180,E1 -9304.677,E2 -9304.677} C_VEL
LIN {X 0,Y 432.343,Z 134.632,A -85,B 0,C 180,E1 -9308.149,E2 -9308.149} C_VEL
LIN {X 0,Y 432.367,Z 134.629,A -85,B 0,C 180,E1 -9311.793,E2 -9311.793} C_VEL
LIN {X 0,Y 432.375,Z 134.624,A -85,B 0,C 180,E1 -9314.341,E2 -9314.341} C_VEL
LIN {X 0,Y 432.363,Z 134.625,A -85,B 0,C 180,E1 -9318.393,E2 -9318.393} C_VEL
LIN {X 0,Y 432.347,Z 134.631,A -85,B 0,C 180,E1 -9321.852,E2 -9321.852} C_VEL
LIN {X 0,Y 432.336,Z 134.631,A -85,B 0,C 180,E1 -9325.323,E2 -9325.323} C_VEL
LIN {X 0,Y 432.318,Z 134.629,A -85,B 0,C 180,E1 -9328.654,E2 -9328.654} C_VEL
LIN {X 0,Y 432.378,Z 134.625,A -85,B 0,C 180,E1 -9331.877,E2 -9331.877} C_VEL
LIN {X 0,Y 432.348,Z 134.628,A -85,B 0,C 180,E1 -9334.999,E2 -9334.999} C_VEL
LIN {X 0,Y 432.354,Z 134.626,A -85,B 0,C 180,E1 -9338.046,E2 -9338.046} C_VEL
LIN {X 0,Y 432.384,Z 134.626,A -85,B 0,C 180,E1 -9341.03,E2 -9341.03} C_VEL
LIN {X 0,Y 432.428,Z 134.616,A -85,B 0,C 180,E1 -9343.961,E2 -9343.961} C_VEL
LIN {X 0,Y 432.457,Z 134.613,A -85,B 0,C 180,E1 -9347.804,E2 -9347.804} C_VEL
LIN {X 0,Y 432.49,Z 134.61,A -85,B 0,C 180,E1 -9351.591,E2 -9351.591} C_VEL
LIN {X 0,Y 432.592,Z 134.597,A -85,B 0,C 180,E1 -9354.406,E2 -9354.406} C_VEL
LIN {X 0,Y 432.604,Z 134.594,A -85,B 0,C 180,E1 -9358.138,E2 -9358.138} C_VEL
LIN {X 0,Y 432.732,Z 134.578,A -85,B 0,C 180,E1 -9360,E2 -9360} C_VEL
LIN {X 0,Y 432.603,Z 134.601,A -85,B 0,C 180,E1 -9362.794,E2 -9362.794} C_VEL
LIN {X 0,Y 432.572,Z 134.603,A -85,B 0,C 180,E1 -9366.531,E2 -9366.531} C_VEL
LIN {X 0,Y 432.442,Z 134.615,A -85,B 0,C 180,E1 -9369.353,E2 -9369.353} C_VEL
LIN {X 0,Y 432.429,Z 134.62,A -85,B 0,C 180,E1 -9372.804,E2 -9372.804} C_VEL
LIN {X 0,Y 432.411,Z 134.625,A -85,B 0,C 180,E1 -9376.479,E2 -9376.479} C_VEL
LIN {X 0,Y 432.338,Z 134.629,A -85,B 0,C 180,E1 -9379.961,E2 -9379.961} C_VEL
LIN {X 0,Y 432.316,Z 134.631,A -85,B 0,C 180,E1 -9382.965,E2 -9382.965} C_VEL
LIN {X 0,Y 432.359,Z 134.628,A -85,B 0,C 180,E1 -9386.033,E2 -9386.033} C_VEL
LIN {X 0,Y 432.342,Z 134.626,A -85,B 0,C 180,E1 -9389.188,E2 -9389.188} C_VEL
LIN {X 0,Y 432.322,Z 134.633,A -85,B 0,C 180,E1 -9392.443,E2 -9392.443} C_VEL
LIN {X 0,Y 432.344,Z 134.628,A -85,B 0,C 180,E1 -9395.632,E2 -9395.632} C_VEL
LIN {X 0,Y 432.357,Z 134.625,A -85,B 0,C 180,E1 -9398.718,E2 -9398.718} C_VEL
LIN {X 0,Y 432.366,Z 134.629,A -85,B 0,C 180,E1 -9401.794,E2 -9401.794} C_VEL
LIN {X 0,Y 432.337,Z 134.63,A -85,B 0,C 180,E1 -9404.347,E2 -9404.347} C_VEL
LIN {X 0,Y 432.32,Z 134.629,A -85,B 0,C 180,E1 -9407.016,E2 -9407.016} C_VEL
LIN {X 0,Y 432.334,Z 134.635,A -85,B 0,C 180,E1 -9409.821,E2 -9409.821} C_VEL
LIN {X 0,Y 432.307,Z 134.631,A -85,B 0,C 180,E1 -9413.023,E2 -9413.023} C_VEL
LIN {X 0,Y 432.36,Z 134.628,A -85,B 0,C 180,E1 -9415.997,E2 -9415.997} C_VEL
LIN {X 0,Y 432.349,Z 134.631,A -85,B 0,C 180,E1 -9419.49,E2 -9419.49} C_VEL
LIN {X 0,Y 432.441,Z 134.668,A -85,B 0,C 180,E1 -9421.98,E2 -9421.98} C_VEL
LIN {X 0,Y 435.213,Z 148.722,A -85,B 0,C 180,E1 -9424.732,E2 -9424.732} C_VEL
LIN {X 0,Y 435.148,Z 153.922,A -85,B 0,C 180,E1 -9425.68,E2 -9425.68} C_VEL
LIN {X 0,Y 434.179,Z 170.53,A -85,B 0,C 180,E1 -9428.642,E2 -9428.642} C_VEL
LIN {X 0,Y 433.441,Z 185.709,A -85,B 0,C 180,E1 -9431.323,E2 -9431.323} C_VEL
LIN {X 0,Y 433.326,Z 188.116,A -85,B 0,C 180,E1 -9431.747,E2 -9431.747} C_VEL
LIN {X 0,Y 436.711,Z 213.312,A -85,B 0,C 180,E1 -9432.358,E2 -9432.358} C_VEL
LIN {X 0,Y 435.663,Z 297.332,A -85,B 0,C 180,E1 -9433.903,E2 -9433.903} C_VEL
LIN {X 0,Y 435.082,Z 311.577,A -85,B 0,C 180,E1 -9434.362,E2 -9434.362} C_VEL
LIN {X 0,Y 434.598,Z 323.738,A -85,B 0,C 180,E1 -9434.945,E2 -9434.945} C_VEL
LIN {X 0,Y 433.919,Z 335.534,A -85,B 0,C 180,E1 -9435.7,E2 -9435.7} C_VEL
LIN {X 0,Y 433.377,Z 346.455,A -85,B 0,C 180,E1 -9436.592,E2 -9436.592} C_VEL
LIN {X 0,Y 432.79,Z 357.295,A -85,B 0,C 180,E1 -9437.694,E2 -9437.694} C_VEL
LIN {X 0,Y 432.271,Z 367.408,A -85,B 0,C 180,E1 -9438.987,E2 -9438.987} C_VEL
LIN {X 0,Y 431.813,Z 376.306,A -85,B 0,C 180,E1 -9440.397,E2 -9440.397} C_VEL
LIN {X 0,Y 431.554,Z 383.388,A -85,B 0,C 180,E1 -9441.808,E2 -9441.808} C_VEL
LIN {X 0,Y 431.337,Z 389.865,A -85,B 0,C 180,E1 -9443.451,E2 -9443.451} C_VEL
LIN {X 0,Y 431.315,Z 394.095,A -85,B 0,C 180,E1 -9444.859,E2 -9444.859} C_VEL
LIN {X 0,Y 431.256,Z 397.215,A -85,B 0,C 180,E1 -9446.263,E2 -9446.263} C_VEL
LIN {X 0,Y 431.33,Z 398.755,A -85,B 0,C 180,E1 -9447.199,E2 -9447.199} C_VEL
LIN {X 0,Y 431.289,Z 399.813,A -85,B 0,C 180,E1 -9448.133,E2 -9448.133} C_VEL
LIN {X 0,Y 431.286,Z 400.463,A -85,B 0,C 180,E1 -9449.067,E2 -9449.067} C_VEL
LIN {X 0,Y 431.294,Z 400.709,A -85,B 0,C 180,E1 -9450,E2 -9450} C_VEL
LIN {X 0,Y 431.257,Z 400.533,A -85,B 0,C 180,E1 -9450.934,E2 -9450.934} C_VEL
LIN {X 0,Y 431.268,Z 399.909,A -85,B 0,C 180,E1 -9451.868,E2 -9451.868} C_VEL
LIN {X 0,Y 431.327,Z 398.883,A -85,B 0,C 180,E1 -9452.802,E2 -9452.802} C_VEL
LIN {X 0,Y 431.238,Z 397.438,A -85,B 0,C 180,E1 -9453.738,E2 -9453.738} C_VEL
LIN {X 0,Y 431.313,Z 394.412,A -85,B 0,C 180,E1 -9455.142,E2 -9455.142} C_VEL
LIN {X 0,Y 431.291,Z 390.31,A -85,B 0,C 180,E1 -9456.55,E2 -9456.55} C_VEL
LIN {X 0,Y 431.563,Z 384.032,A -85,B 0,C 180,E1 -9458.192,E2 -9458.192} C_VEL
LIN {X 0,Y 431.822,Z 377.163,A -85,B 0,C 180,E1 -9459.603,E2 -9459.603} C_VEL
LIN {X 0,Y 432.299,Z 368.658,A -85,B 0,C 180,E1 -9461.013,E2 -9461.013} C_VEL
LIN {X 0,Y 432.842,Z 359.951,A -85,B 0,C 180,E1 -9462.186,E2 -9462.186} C_VEL
LIN {X 0,Y 433.409,Z 349.247,A -85,B 0,C 180,E1 -9463.359,E2 -9463.359} C_VEL
LIN {X 0,Y 434.202,Z 337.205,A -85,B 0,C 180,E1 -9464.41,E2 -9464.41} C_VEL
LIN {X 0,Y 434.92,Z 325.133,A -85,B 0,C 180,E1 -9465.224,E2 -9465.224} C_VEL
LIN {X 0,Y 435.556,Z 312.697,A -85,B 0,C 180,E1 -9465.861,E2 -9465.861} C_VEL
LIN {X 0,Y 436.161,Z 300.005,A -85,B 0,C 180,E1 -9466.319,E2 -9466.319} C_VEL
LIN {X 0,Y 436.493,Z 284.107,A -85,B 0,C 180,E1 -9466.667,E2 -9466.667} C_VEL
LIN {X 0,Y 437.482,Z 212.721,A -85,B 0,C 180,E1 -9468.012,E2 -9468.012} C_VEL
LIN {X 0,Y 434.793,Z 193.151,A -85,B 0,C 180,E1 -9468.54,E2 -9468.54} C_VEL
LIN {X 0,Y 433.512,Z 185.701,A -85,B 0,C 180,E1 -9468.772,E2 -9468.772} C_VEL
LIN {X 0,Y 434.416,Z 168.084,A -85,B 0,C 180,E1 -9471.845,E2 -9471.845} C_VEL
LIN {X 0,Y 435.424,Z 149.566,A -85,B 0,C 180,E1 -9475.131,E2 -9475.131} C_VEL
LIN {X 0,Y 433.705,Z 140.12,A -85,B 0,C 180,E1 -9476.983,E2 -9476.983} C_VEL
LIN {X 0,Y 432.419,Z 134.629,A -85,B 0,C 180,E1 -9478.121,E2 -9478.121} C_VEL
LIN {X 0,Y 432.325,Z 134.636,A -85,B 0,C 180,E1 -9481.346,E2 -9481.346} C_VEL
LIN {X 0,Y 432.343,Z 134.632,A -85,B 0,C 180,E1 -9484.677,E2 -9484.677} C_VEL
LIN {X 0,Y 432.343,Z 134.633,A -85,B 0,C 180,E1 -9488.15,E2 -9488.15} C_VEL
LIN {X 0,Y 432.337,Z 134.633,A -85,B 0,C 180,E1 -9491.602,E2 -9491.602} C_VEL
LIN {X 0,Y 432.337,Z 134.632,A -85,B 0,C 180,E1 -9494.347,E2 -9494.347} C_VEL
LIN {X 0,Y 432.324,Z 134.63,A -85,B 0,C 180,E1 -9497.016,E2 -9497.016} C_VEL
LIN {X 0,Y 432.337,Z 134.631,A -85,B 0,C 180,E1 -9499.821,E2 -9499.821} C_VEL
LIN {X 0,Y 432.309,Z 134.631,A -85,B 0,C 180,E1 -9503.022,E2 -9503.022} C_VEL
LIN {X 0,Y 432.361,Z 134.624,A -85,B 0,C 180,E1 -9505.997,E2 -9505.997} C_VEL
LIN {X 0,Y 432.35,Z 134.629,A -85,B 0,C 180,E1 -9509.49,E2 -9509.49} C_VEL
LIN {X 0,Y 432.394,Z 134.624,A -85,B 0,C 180,E1 -9512.928,E2 -9512.928} C_VEL
LIN {X 0,Y 432.373,Z 134.624,A -85,B 0,C 180,E1 -9516.023,E2 -9516.023} C_VEL
LIN {X 0,Y 432.353,Z 134.629,A -85,B 0,C 180,E1 -9519.046,E2 -9519.046} C_VEL
LIN {X 0,Y 432.362,Z 134.622,A -85,B 0,C 180,E1 -9522.01,E2 -9522.01} C_VEL
LIN {X 0,Y 432.397,Z 134.624,A -85,B 0,C 180,E1 -9524.926,E2 -9524.926} C_VEL
LIN {X 0,Y 432.462,Z 134.614,A -85,B 0,C 180,E1 -9527.803,E2 -9527.803} C_VEL
LIN {X 0,Y 432.466,Z 134.615,A -85,B 0,C 180,E1 -9531.589,E2 -9531.589} C_VEL
LIN {X 0,Y 432.588,Z 134.603,A -85,B 0,C 180,E1 -9534.406,E2 -9534.406} C_VEL
LIN {X 0,Y 432.605,Z 134.602,A -85,B 0,C 180,E1 -9538.138,E2 -9538.138} C_VEL
LIN {X 0,Y 432.73,Z 134.584,A -85,B 0,C 180,E1 -9540,E2 -9540} C_VEL
LIN {X 0,Y 432.58,Z 134.604,A -85,B 0,C 180,E1 -9542.793,E2 -9542.793} C_VEL
LIN {X 0,Y 432.414,Z 134.815,A -85,B 0,C 180,E1 -9544.136,E2 -9544.136} C_VEL
LIN {X 0,Y 434.257,Z 143.037,A -85,B 0,C 180,E1 -9546.038,E2 -9546.038} C_VEL
LIN {X 0,Y 434.445,Z 144.675,A -85,B 0,C 180,E1 -9546.356,E2 -9546.356} C_VEL
LIN {X 0,Y 438.186,Z 160.399,A -85,B 0,C 180,E1 -9546.88,E2 -9546.88} C_VEL
LIN {X 0,Y 436.656,Z 252.416,A -85,B 0,C 180,E1 -9548.649,E2 -9548.649} C_VEL
LIN {X 0,Y 436.325,Z 265.635,A -85,B 0,C 180,E1 -9549.094,E2 -9549.094} C_VEL
LIN {X 0,Y 435.912,Z 277.447,A -85,B 0,C 180,E1 -9549.665,E2 -9549.665} C_VEL
LIN {X 0,Y 435.33,Z 289.734,A -85,B 0,C 180,E1 -9550.464,E2 -9550.464} C_VEL
LIN {X 0,Y 434.673,Z 301.231,A -85,B 0,C 180,E1 -9551.423,E2 -9551.423} C_VEL
LIN {X 0,Y 434.051,Z 311.543,A -85,B 0,C 180,E1 -9552.507,E2 -9552.507} C_VEL
LIN {X 0,Y 433.467,Z 320.6,A -85,B 0,C 180,E1 -9553.684,E2 -9553.684} C_VEL
LIN {X 0,Y 432.89,Z 329.186,A -85,B 0,C 180,E1 -9555.056,E2 -9555.056} C_VEL
LIN {X 0,Y 432.395,Z 336.289,A -85,B 0,C 180,E1 -9556.47,E2 -9556.47} C_VEL
LIN {X 0,Y 432.016,Z 342.326,A -85,B 0,C 180,E1 -9558.004,E2 -9558.004} C_VEL
LIN {X 0,Y 431.745,Z 346.173,A -85,B 0,C 180,E1 -9559.242,E2 -9559.242} C_VEL
LIN {X 0,Y 431.475,Z 350.162,A -85,B 0,C 180,E1 -9560.998,E2 -9560.998} C_VEL
LIN {X 0,Y 431.36,Z 351.768,A -85,B 0,C 180,E1 -9562.007,E2 -9562.007} C_VEL
LIN {X 0,Y 431.241,Z 352.846,A -85,B 0,C 180,E1 -9563.025,E2 -9563.025} C_VEL
LIN {X 0,Y 431.216,Z 353.504,A -85,B 0,C 180,E1 -9564.119,E2 -9564.119} C_VEL
LIN {X 0,Y 431.184,Z 353.59,A -85,B 0,C 180,E1 -9565.073,E2 -9565.073} C_VEL
LIN {X 0,Y 431.212,Z 353.088,A -85,B 0,C 180,E1 -9566.31,E2 -9566.31} C_VEL
LIN {X 0,Y 431.252,Z 352.34,A -85,B 0,C 180,E1 -9567.149,E2 -9567.149} C_VEL
LIN {X 0,Y 431.313,Z 350.623,A -85,B 0,C 180,E1 -9568.369,E2 -9568.369} C_VEL
LIN {X 0,Y 431.525,Z 347.725,A -85,B 0,C 180,E1 -9569.784,E2 -9569.784} C_VEL
LIN {X 0,Y 431.678,Z 343.15,A -85,B 0,C 180,E1 -9571.398,E2 -9571.398} C_VEL
LIN {X 0,Y 432.083,Z 336.928,A -85,B 0,C 180,E1 -9573.017,E2 -9573.017} C_VEL
LIN {X 0,Y 432.424,Z 329.808,A -85,B 0,C 180,E1 -9574.474,E2 -9574.474} C_VEL
LIN {X 0,Y 432.914,Z 321.997,A -85,B 0,C 180,E1 -9575.762,E2 -9575.762} C_VEL
LIN {X 0,Y 433.32,Z 313.787,A -85,B 0,C 180,E1 -9576.877,E2 -9576.877} C_VEL
LIN {X 0,Y 433.877,Z 303.738,A -85,B 0,C 180,E1 -9577.99,E2 -9577.99} C_VEL
LIN {X 0,Y 434.451,Z 292.558,A -85,B 0,C 180,E1 -9578.989,E2 -9578.989} C_VEL
LIN {X 0,Y 434.959,Z 280.903,A -85,B 0,C 180,E1 -9579.81,E2 -9579.81} C_VEL
LIN {X 0,Y 435.421,Z 268.085,A -85,B 0,C 180,E1 -9580.49,E2 -9580.49} C_VEL
LIN {X 0,Y 435.687,Z 254.813,A -85,B 0,C 180,E1 -9580.991,E2 -9580.991} C_VEL
LIN {X 0,Y 435.973,Z 240.358,A -85,B 0,C 180,E1 -9581.311,E2 -9581.311} C_VEL
LIN {X 0,Y 437.021,Z 159.386,A -85,B 0,C 180,E1 -9582.782,E2 -9582.782} C_VEL
LIN {X 0,Y 433.616,Z 142.562,A -85,B 0,C 180,E1 -9583.249,E2 -9583.249} C_VEL
LIN {X 0,Y 432.424,Z 134.622,A -85,B 0,C 180,E1 -9585.092,E2 -9585.092} C_VEL
LIN {X 0,Y 432.332,Z 134.629,A -85,B 0,C 180,E1 -9588.398,E2 -9588.398} C_VEL
LIN {X 0,Y 432.334,Z 134.632,A -85,B 0,C 180,E1 -9591.849,E2 -9591.849} C_VEL
LIN {X 0,Y 432.337,Z 134.632,A -85,B 0,C 180,E1 -9595.322,E2 -9595.322} C_VEL
LIN {X 0,Y 432.323,Z 134.634,A -85,B 0,C 180,E1 -9597.702,E2 -9597.702} C_VEL
LIN {X 0,Y 431.676,Z 134.71,A -85,B 0,C 180,E1 -9598.48,E2 -9598.48} C_VEL
LIN {X 0,Y 428.837,Z 135.067,A -85,B 0,C 180,E1 -9599.744,E2 -9599.744} C_VEL
LIN {X 0,Y 426.428,Z 135.369,A -85,B 0,C 180,E1 -9600.765,E2 -9600.765} C_VEL
LIN {X 0,Y 425.399,Z 135.497,A -85,B 0,C 180,E1 -9601.553,E2 -9601.553} C_VEL
LIN {X 0,Y 425.32,Z 135.503,A -85,B 0,C 180,E1 -9601.82,E2 -9601.82} C_VEL
LIN {X 0,Y 425.294,Z 135.505,A -85,B 0,C 180,E1 -9604.554,E2 -9604.554} C_VEL
LIN {X 0,Y 425.287,Z 135.508,A -85,B 0,C 180,E1 -9607.661,E2 -9607.661} C_VEL
LIN {X 0,Y 425.36,Z 135.498,A -85,B 0,C 180,E1 -9610.704,E2 -9610.704} C_VEL
LIN {X 0,Y 425.387,Z 135.495,A -85,B 0,C 180,E1 -9613.688,E2 -9613.688} C_VEL
LIN {X 0,Y 425.411,Z 135.492,A -85,B 0,C 180,E1 -9617.598,E2 -9617.598} C_VEL
LIN {X 0,Y 425.441,Z 135.488,A -85,B 0,C 180,E1 -9621.45,E2 -9621.45} C_VEL
LIN {X 0,Y 425.549,Z 135.474,A -85,B 0,C 180,E1 -9624.313,E2 -9624.313} C_VEL
LIN {X 0,Y 425.575,Z 135.47,A -85,B 0,C 180,E1 -9628.107,E2 -9628.107} C_VEL
LIN {X 0,Y 425.702,Z 135.454,A -85,B 0,C 180,E1 -9630,E2 -9630} C_VEL
LIN {X 0,Y 425.554,Z 135.478,A -85,B 0,C 180,E1 -9632.84,E2 -9632.84} C_VEL
LIN {X 0,Y 425.522,Z 135.483,A -85,B 0,C 180,E1 -9636.639,E2 -9636.639} C_VEL
LIN {X 0,Y 425.4,Z 135.491,A -85,B 0,C 180,E1 -9639.509,E2 -9639.509} C_VEL
LIN {X 0,Y 425.391,Z 135.495,A -85,B 0,C 180,E1 -9642.903,E2 -9642.903} C_VEL
LIN {X 0,Y 425.359,Z 135.502,A -85,B 0,C 180,E1 -9646.605,E2 -9646.605} C_VEL
LIN {X 0,Y 425.326,Z 135.501,A -85,B 0,C 180,E1 -9649.636,E2 -9649.636} C_VEL
LIN {X 0,Y 425.285,Z 135.513,A -85,B 0,C 180,E1 -9652.338,E2 -9652.338} C_VEL
LIN {X 0,Y 425.287,Z 135.505,A -85,B 0,C 180,E1 -9655.445,E2 -9655.445} C_VEL
LIN {X 0,Y 425.335,Z 135.502,A -85,B 0,C 180,E1 -9658.631,E2 -9658.631} C_VEL
LIN {X 0,Y 425.27,Z 135.512,A -85,B 0,C 180,E1 -9661.926,E2 -9661.926} C_VEL
LIN {X 0,Y 425.297,Z 135.505,A -85,B 0,C 180,E1 -9665.336,E2 -9665.336} C_VEL
LIN {X 0,Y 425.31,Z 135.502,A -85,B 0,C 180,E1 -9668.897,E2 -9668.897} C_VEL
LIN {X 0,Y 425.327,Z 135.501,A -85,B 0,C 180,E1 -9672.646,E2 -9672.646} C_VEL
LIN {X 0,Y 425.291,Z 135.506,A -85,B 0,C 180,E1 -9675.282,E2 -9675.282} C_VEL
LIN {X 0,Y 425.3,Z 135.504,A -85,B 0,C 180,E1 -9678.625,E2 -9678.625} C_VEL
LIN {X 0,Y 425.318,Z 135.503,A -85,B 0,C 180,E1 -9681.104,E2 -9681.104} C_VEL
LIN {X 0,Y 425.296,Z 135.504,A -85,B 0,C 180,E1 -9684.664,E2 -9684.664} C_VEL
LIN {X 0,Y 425.262,Z 135.51,A -85,B 0,C 180,E1 -9688.073,E2 -9688.073} C_VEL
LIN {X 0,Y 425.328,Z 135.506,A -85,B 0,C 180,E1 -9691.368,E2 -9691.368} C_VEL
LIN {X 0,Y 425.292,Z 135.505,A -85,B 0,C 180,E1 -9694.555,E2 -9694.555} C_VEL
LIN {X 0,Y 425.285,Z 135.509,A -85,B 0,C 180,E1 -9697.661,E2 -9697.661} C_VEL
LIN {X 0,Y 425.359,Z 135.498,A -85,B 0,C 180,E1 -9700.704,E2 -9700.704} C_VEL
LIN {X 0,Y 425.386,Z 135.495,A -85,B 0,C 180,E1 -9703.689,E2 -9703.689} C_VEL
LIN {X 0,Y 425.409,Z 135.492,A -85,B 0,C 180,E1 -9707.598,E2 -9707.598} C_VEL
LIN {X 0,Y 425.44,Z 135.489,A -85,B 0,C 180,E1 -9711.45,E2 -9711.45} C_VEL
LIN {X 0,Y 425.548,Z 135.473,A -85,B 0,C 180,E1 -9714.314,E2 -9714.314} C_VEL
LIN {X 0,Y 425.574,Z 135.47,A -85,B 0,C 180,E1 -9718.108,E2 -9718.108} C_VEL
LIN {X 0,Y 425.701,Z 135.454,A -85,B 0,C 180,E1 -9720,E2 -9720} C_VEL
LIN {X 0,Y 425.554,Z 135.479,A -85,B 0,C 180,E1 -9722.84,E2 -9722.84} C_VEL
LIN {X 0,Y 425.53,Z 135.481,A -85,B 0,C 180,E1 -9726.639,E2 -9726.639} C_VEL
LIN {X 0,Y 425.4,Z 135.491,A -85,B 0,C 180,E1 -9729.51,E2 -9729.51} C_VEL
LIN {X 0,Y 425.392,Z 135.496,A -85,B 0,C 180,E1 -9732.904,E2 -9732.904} C_VEL
LIN {X 0,Y 425.36,Z 135.502,A -85,B 0,C 180,E1 -9736.606,E2 -9736.606} C_VEL
LIN {X 0,Y 425.327,Z 135.5,A -85,B 0,C 180,E1 -9739.636,E2 -9739.636} C_VEL
LIN {X 0,Y 425.286,Z 135.512,A -85,B 0,C 180,E1 -9742.339,E2 -9742.339} C_VEL
LIN {X 0,Y 425.289,Z 135.505,A -85,B 0,C 180,E1 -9745.446,E2 -9745.446} C_VEL
LIN {X 0,Y 425.347,Z 135.498,A -85,B 0,C 180,E1 -9747.558,E2 -9747.558} C_VEL
LIN {X 0,Y 425.287,Z 135.506,A -85,B 0,C 180,E1 -9750.817,E2 -9750.817} C_VEL
LIN {X 0,Y 425.311,Z 135.508,A -85,B 0,C 180,E1 -9754.288,E2 -9754.288} C_VEL
LIN {X 0,Y 425.287,Z 135.508,A -85,B 0,C 180,E1 -9757.694,E2 -9757.694} C_VEL
LIN {X 0,Y 425.298,Z 135.506,A -85,B 0,C 180,E1 -9760.524,E2 -9760.524} C_VEL
LIN {X 0,Y 425.258,Z 135.51,A -85,B 0,C 180,E1 -9763.352,E2 -9763.352} C_VEL
LIN {X 0,Y 425.258,Z 135.509,A -85,B 0,C 180,E1 -9766.65,E2 -9766.65} C_VEL
LIN {X 0,Y 425.287,Z 135.512,A -85,B 0,C 180,E1 -9769.873,E2 -9769.873} C_VEL
LIN {X 0,Y 425.278,Z 135.507,A -85,B 0,C 180,E1 -9772.489,E2 -9772.489} C_VEL
LIN {X 0,Y 425.308,Z 135.508,A -85,B 0,C 180,E1 -9775.818,E2 -9775.818} C_VEL
LIN {X 0,Y 425.292,Z 135.51,A -85,B 0,C 180,E1 -9779.239,E2 -9779.239} C_VEL
LIN {X 0,Y 425.383,Z 135.638,A -85,B 0,C 180,E1 -9781.776,E2 -9781.776} C_VEL
LIN {X 0,Y 428.159,Z 149.442,A -85,B 0,C 180,E1 -9784.529,E2 -9784.529} C_VEL
LIN {X 0,Y 428.29,Z 153.358,A -85,B 0,C 180,E1 -9785.264,E2 -9785.264} C_VEL
LIN {X 0,Y 427.27,Z 169.98,A -85,B 0,C 180,E1 -9788.279,E2 -9788.279} C_VEL
LIN {X 0,Y 426.494,Z 185.163,A -85,B 0,C 180,E1 -9791.008,E2 -9791.008} C_VEL
LIN {X 0,Y 426.334,Z 187.933,A -85,B 0,C 180,E1 -9791.483,E2 -9791.483} C_VEL
LIN {X 0,Y 429.865,Z 214.388,A -85,B 0,C 180,E1 -9792.129,E2 -9792.129} C_VEL
LIN {X 0,Y 428.761,Z 297.512,A -85,B 0,C 180,E1 -9793.698,E2 -9793.698} C_VEL
LIN {X 0,Y 428.155,Z 311.558,A -85,B 0,C 180,E1 -9794.164,E2 -9794.164} C_VEL
LIN {X 0,Y 427.633,Z 323.598,A -85,B 0,C 180,E1 -9794.755,E2 -9794.755} C_VEL
LIN {X 0,Y 426.894,Z 336.141,A -85,B 0,C 180,E1 -9795.582,E2 -9795.582} C_VEL
LIN {X 0,Y 426.356,Z 346.598,A -85,B 0,C 180,E1 -9796.461,E2 -9796.461} C_VEL
LIN {X 0,Y 425.781,Z 356.575,A -85,B 0,C 180,E1 -9797.493,E2 -9797.493} C_VEL
LIN {X 0,Y 425.357,Z 365.069,A -85,B 0,C 180,E1 -9798.564,E2 -9798.564} C_VEL
LIN {X 0,Y 424.793,Z 374.303,A -85,B 0,C 180,E1 -9799.996,E2 -9799.996} C_VEL
LIN {X 0,Y 424.514,Z 381.746,A -85,B 0,C 180,E1 -9801.431,E2 -9801.431} C_VEL
LIN {X 0,Y 424.319,Z 387.687,A -85,B 0,C 180,E1 -9802.865,E2 -9802.865} C_VEL
LIN {X 0,Y 424.182,Z 392.335,A -85,B 0,C 180,E1 -9804.295,E2 -9804.295} C_VEL
LIN {X 0,Y 424.211,Z 394.775,A -85,B 0,C 180,E1 -9805.249,E2 -9805.249} C_VEL
LIN {X 0,Y 424.161,Z 396.759,A -85,B 0,C 180,E1 -9806.2,E2 -9806.2} C_VEL
LIN {X 0,Y 424.257,Z 398.319,A -85,B 0,C 180,E1 -9807.152,E2 -9807.152} C_VEL
LIN {X 0,Y 424.211,Z 399.395,A -85,B 0,C 180,E1 -9808.102,E2 -9808.102} C_VEL
LIN {X 0,Y 424.199,Z 400.054,A -85,B 0,C 180,E1 -9809.051,E2 -9809.051} C_VEL
LIN {X 0,Y 424.217,Z 400.311,A -85,B 0,C 180,E1 -9810,E2 -9810} C_VEL
LIN {X 0,Y 424.172,Z 400.15,A -85,B 0,C 180,E1 -9810.95,E2 -9810.95} C_VEL
LIN {X 0,Y 424.192,Z 399.537,A -85,B 0,C 180,E1 -9811.899,E2 -9811.899} C_VEL
LIN {X 0,Y 424.235,Z 398.516,A -85,B 0,C 180,E1 -9812.849,E2 -9812.849} C_VEL
LIN {X 0,Y 424.144,Z 397.078,A -85,B 0,C 180,E1 -9813.801,E2 -9813.801} C_VEL
LIN {X 0,Y 424.219,Z 394.068,A -85,B 0,C 180,E1 -9815.228,E2 -9815.228} C_VEL
LIN {X 0,Y 424.225,Z 389.983,A -85,B 0,C 180,E1 -9816.66,E2 -9816.66} C_VEL
LIN {X 0,Y 424.492,Z 383.727,A -85,B 0,C 180,E1 -9818.33,E2 -9818.33} C_VEL
LIN {X 0,Y 424.793,Z 376.875,A -85,B 0,C 180,E1 -9819.764,E2 -9819.764} C_VEL
LIN {X 0,Y 425.314,Z 368.399,A -85,B 0,C 180,E1 -9821.196,E2 -9821.196} C_VEL
LIN {X 0,Y 425.861,Z 359.739,A -85,B 0,C 180,E1 -9822.389,E2 -9822.389} C_VEL
LIN {X 0,Y 426.476,Z 349.305,A -85,B 0,C 180,E1 -9823.557,E2 -9823.557} C_VEL
LIN {X 0,Y 427.31,Z 337.109,A -85,B 0,C 180,E1 -9824.648,E2 -9824.648} C_VEL
LIN {X 0,Y 428.072,Z 325.168,A -85,B 0,C 180,E1 -9825.474,E2 -9825.474} C_VEL
LIN {X 0,Y 428.756,Z 312.904,A -85,B 0,C 180,E1 -9826.119,E2 -9826.119} C_VEL
LIN {X 0,Y 429.412,Z 299.641,A -85,B 0,C 180,E1 -9826.613,E2 -9826.613} C_VEL
LIN {X 0,Y 429.772,Z 283.916,A -85,B 0,C 180,E1 -9826.966,E2 -9826.966} C_VEL
LIN {X 0,Y 430.8,Z 213.303,A -85,B 0,C 180,E1 -9828.33,E2 -9828.33} C_VEL
LIN {X 0,Y 428.088,Z 193.608,A -85,B 0,C 180,E1 -9828.881,E2 -9828.881} C_VEL
LIN {X 0,Y 426.63,Z 185.288,A -85,B 0,C 180,E1 -9829.139,E2 -9829.139} C_VEL
LIN {X 0,Y 427.592,Z 167.982,A -85,B 0,C 180,E1 -9832.212,E2 -9832.212} C_VEL
LIN {X 0,Y 428.569,Z 151.247,A -85,B 0,C 180,E1 -9835.238,E2 -9835.238} C_VEL
LIN {X 0,Y 426.755,Z 141.397,A -85,B 0,C 180,E1 -9837.214,E2 -9837.214} C_VEL
LIN {X 0,Y 425.348,Z 135.511,A -85,B 0,C 180,E1 -9838.497,E2 -9838.497} C_VEL
LIN {X 0,Y 425.269,Z 135.517,A -85,B 0,C 180,E1 -9841.927,E2 -9841.927} C_VEL
LIN {X 0,Y 425.303,Z 135.507,A -85,B 0,C 180,E1 -9845.336,E2 -9845.336} C_VEL
LIN {X 0,Y 425.304,Z 135.507,A -85,B 0,C 180,E1 -9849.044,E2 -9849.044} C_VEL
LIN {X 0,Y 425.278,Z 135.51,A -85,B 0,C 180,E1 -9852.653,E2 -9852.653} C_VEL
LIN {X 0,Y 425.265,Z 135.511,A -85,B 0,C 180,E1 -9856.044,E2 -9856.044} C_VEL
LIN {X 0,Y 425.277,Z 135.504,A -85,B 0,C 180,E1 -9858.621,E2 -9858.621} C_VEL
LIN {X 0,Y 425.3,Z 135.502,A -85,B 0,C 180,E1 -9861.101,E2 -9861.101} C_VEL
LIN {X 0,Y 425.301,Z 135.503,A -85,B 0,C 180,E1 -9864.664,E2 -9864.664} C_VEL
LIN {X 0,Y 425.267,Z 135.506,A -85,B 0,C 180,E1 -9868.073,E2 -9868.073} C_VEL
LIN {X 0,Y 425.334,Z 135.502,A -85,B 0,C 180,E1 -9871.368,E2 -9871.368} C_VEL
LIN {X 0,Y 425.357,Z 135.499,A -85,B 0,C 180,E1 -9873.505,E2 -9873.505} C_VEL
LIN {X 0,Y 425.31,Z 135.505,A -85,B 0,C 180,E1 -9876.635,E2 -9876.635} C_VEL
LIN {X 0,Y 425.331,Z 135.501,A -85,B 0,C 180,E1 -9880.364,E2 -9880.364} C_VEL
LIN {X 0,Y 425.391,Z 135.494,A -85,B 0,C 180,E1 -9883.688,E2 -9883.688} C_VEL
LIN {X 0,Y 425.415,Z 135.493,A -85,B 0,C 180,E1 -9887.598,E2 -9887.598} C_VEL
LIN {X 0,Y 425.411,Z 135.495,A -85,B 0,C 180,E1 -9891.449,E2 -9891.449} C_VEL
LIN {X 0,Y 425.544,Z 135.48,A -85,B 0,C 180,E1 -9894.313,E2 -9894.313} C_VEL
LIN {X 0,Y 425.574,Z 135.478,A -85,B 0,C 180,E1 -9898.107,E2 -9898.107} C_VEL
LIN {X 0,Y 425.7,Z 135.46,A -85,B 0,C 180,E1 -9900,E2 -9900} C_VEL
LIN {X 0,Y 425.534,Z 135.482,A -85,B 0,C 180,E1 -9902.84,E2 -9902.84} C_VEL
LIN {X 0,Y 425.336,Z 135.667,A -85,B 0,C 180,E1 -9903.789,E2 -9903.789} C_VEL
LIN {X 0,Y 427.417,Z 144.848,A -85,B 0,C 180,E1 -9905.957,E2 -9905.957} C_VEL
LIN {X 0,Y 429.835,Z 153.713,A -85,B 0,C 180,E1 -9906.292,E2 -9906.292} C_VEL
LIN {X 0,Y 431.646,Z 162.31,A -85,B 0,C 180,E1 -9906.574,E2 -9906.574} C_VEL
LIN {X 0,Y 429.939,Z 252.464,A -85,B 0,C 180,E1 -9908.341,E2 -9908.341} C_VEL
LIN {X 0,Y 429.614,Z 265.736,A -85,B 0,C 180,E1 -9908.792,E2 -9908.792} C_VEL
LIN {X 0,Y 429.122,Z 278.577,A -85,B 0,C 180,E1 -9909.426,E2 -9909.426} C_VEL
LIN {X 0,Y 428.507,Z 290.727,A -85,B 0,C 180,E1 -9910.24,E2 -9910.24} C_VEL
LIN {X 0,Y 427.802,Z 302.471,A -85,B 0,C 180,E1 -9911.249,E2 -9911.249} C_VEL
LIN {X 0,Y 427.152,Z 312.584,A -85,B 0,C 180,E1 -9912.35,E2 -9912.35} C_VEL
LIN {X 0,Y 426.521,Z 321.551,A -85,B 0,C 180,E1 -9913.547,E2 -9913.547} C_VEL
LIN {X 0,Y 425.946,Z 329.356,A -85,B 0,C 180,E1 -9914.817,E2 -9914.817} C_VEL
LIN {X 0,Y 425.395,Z 336.76,A -85,B 0,C 180,E1 -9916.311,E2 -9916.311} C_VEL
LIN {X 0,Y 425.001,Z 342.59,A -85,B 0,C 180,E1 -9917.813,E2 -9917.813} C_VEL
LIN {X 0,Y 424.659,Z 347.265,A -85,B 0,C 180,E1 -9919.38,E2 -9919.38} C_VEL
LIN {X 0,Y 424.502,Z 349.515,A -85,B 0,C 180,E1 -9920.345,E2 -9920.345} C_VEL
LIN {X 0,Y 424.285,Z 352.184,A -85,B 0,C 180,E1 -9921.935,E2 -9921.935} C_VEL
LIN {X 0,Y 424.137,Z 353.61,A -85,B 0,C 180,E1 -9923.433,E2 -9923.433} C_VEL
LIN {X 0,Y 424.13,Z 353.972,A -85,B 0,C 180,E1 -9924.472,E2 -9924.472} C_VEL
LIN {X 0,Y 424.098,Z 353.88,A -85,B 0,C 180,E1 -9925.522,E2 -9925.522} C_VEL
LIN {X 0,Y 424.146,Z 353.257,A -85,B 0,C 180,E1 -9926.576,E2 -9926.576} C_VEL
LIN {X 0,Y 424.169,Z 352.121,A -85,B 0,C 180,E1 -9927.64,E2 -9927.64} C_VEL
LIN {X 0,Y 424.355,Z 349.412,A -85,B 0,C 180,E1 -9929.246,E2 -9929.246} C_VEL
LIN {X 0,Y 424.579,Z 345.342,A -85,B 0,C 180,E1 -9930.873,E2 -9930.873} C_VEL
LIN {X 0,Y 424.837,Z 339.912,A -85,B 0,C 180,E1 -9932.468,E2 -9932.468} C_VEL
LIN {X 0,Y 425.188,Z 333.653,A -85,B 0,C 180,E1 -9933.907,E2 -9933.907} C_VEL
LIN {X 0,Y 425.667,Z 326.118,A -85,B 0,C 180,E1 -9935.3,E2 -9935.3} C_VEL
LIN {X 0,Y 426.203,Z 316.578,A -85,B 0,C 180,E1 -9936.709,E2 -9936.709} C_VEL
LIN {X 0,Y 426.789,Z 306.54,A -85,B 0,C 180,E1 -9937.904,E2 -9937.904} C_VEL
LIN {X 0,Y 427.375,Z 295.65,A -85,B 0,C 180,E1 -9938.944,E2 -9938.944} C_VEL
LIN {X 0,Y 427.885,Z 283.879,A -85,B 0,C 180,E1 -9939.834,E2 -9939.834} C_VEL
LIN {X 0,Y 428.42,Z 271.678,A -85,B 0,C 180,E1 -9940.543,E2 -9940.543} C_VEL
LIN {X 0,Y 428.737,Z 258.736,A -85,B 0,C 180,E1 -9941.085,E2 -9941.085} C_VEL
LIN {X 0,Y 429.043,Z 244.645,A -85,B 0,C 180,E1 -9941.459,E2 -9941.459} C_VEL
LIN {X 0,Y 430.203,Z 160.352,A -85,B 0,C 180,E1 -9943.024,E2 -9943.024} C_VEL
LIN {X 0,Y 426.597,Z 142.894,A -85,B 0,C 180,E1 -9943.519,E2 -9943.519} C_VEL
LIN {X 0,Y 425.347,Z 135.504,A -85,B 0,C 180,E1 -9945.274,E2 -9945.274} C_VEL
LIN {X 0,Y 425.273,Z 135.507,A -85,B 0,C 180,E1 -9948.621,E2 -9948.621} C_VEL
LIN {X 0,Y 425.296,Z 135.506,A -85,B 0,C 180,E1 -9951.101,E2 -9951.101} C_VEL
LIN {X 0,Y 425.297,Z 135.504,A -85,B 0,C 180,E1 -9954.664,E2 -9954.664} C_VEL
LIN {X 0,Y 425.263,Z 135.51,A -85,B 0,C 180,E1 -9958.073,E2 -9958.073} C_VEL
LIN {X 0,Y 425.33,Z 135.507,A -85,B 0,C 180,E1 -9961.367,E2 -9961.367} C_VEL
LIN {X 0,Y 425.32,Z 135.503,A -85,B 0,C 180,E1 -9961.82,E2 -9961.82} C_VEL
LIN {X 0,Y 424.656,Z 135.585,A -85,B 0,C 180,E1 -9962.61,E2 -9962.61} C_VEL
LIN {X 0,Y 421.787,Z 135.943,A -85,B 0,C 180,E1 -9963.894,E2 -9963.894} C_VEL
LIN {X 0,Y 419.368,Z 136.245,A -85,B 0,C 180,E1 -9964.93,E2 -9964.93} C_VEL
LIN {X 0,Y 418.348,Z 136.372,A -85,B 0,C 180,E1 -9965.731,E2 -9965.731} C_VEL
LIN {X 0,Y 418.276,Z 136.378,A -85,B 0,C 180,E1 -9966.002,E2 -9966.002} C_VEL
LIN {X 0,Y 418.249,Z 136.388,A -85,B 0,C 180,E1 -9969.337,E2 -9969.337} C_VEL
LIN {X 0,Y 418.279,Z 136.379,A -85,B 0,C 180,E1 -9972.395,E2 -9972.395} C_VEL
LIN {X 0,Y 418.302,Z 136.379,A -85,B 0,C 180,E1 -9975.403,E2 -9975.403} C_VEL
LIN {X 0,Y 418.315,Z 136.374,A -85,B 0,C 180,E1 -9978.369,E2 -9978.369} C_VEL
LIN {X 0,Y 418.483,Z 136.353,A -85,B 0,C 180,E1 -9982.279,E2 -9982.279} C_VEL
LIN {X 0,Y 418.508,Z 136.35,A -85,B 0,C 180,E1 -9984.217,E2 -9984.217} C_VEL
LIN {X 0,Y 418.544,Z 136.346,A -85,B 0,C 180,E1 -9988.075,E2 -9988.075} C_VEL
LIN {X 0,Y 418.671,Z 136.33,A -85,B 0,C 180,E1 -9990,E2 -9990} C_VEL
LIN {X 0,Y 418.508,Z 136.355,A -85,B 0,C 180,E1 -9992.887,E2 -9992.887} C_VEL
LIN {X 0,Y 418.486,Z 136.359,A -85,B 0,C 180,E1 -9996.751,E2 -9996.751} C_VEL
LIN {X 0,Y 418.34,Z 136.371,A -85,B 0,C 180,E1 -9999.671,E2 -9999.671} C_VEL
LIN {X 0,Y 418.344,Z 136.372,A -85,B 0,C 180,E1 -10003.001,E2 -10003.001} C_VEL
LIN {X 0,Y 418.311,Z 136.378,A -85,B 0,C 180,E1 -10006.735,E2 -10006.735} C_VEL
LIN {X 0,Y 418.268,Z 136.381,A -85,B 0,C 180,E1 -10009.79,E2 -10009.79} C_VEL
LIN {X 0,Y 418.229,Z 136.387,A -85,B 0,C 180,E1 -10012.736,E2 -10012.736} C_VEL
LIN {X 0,Y 418.265,Z 136.383,A -85,B 0,C 180,E1 -10015.904,E2 -10015.904} C_VEL
LIN {X 0,Y 418.271,Z 136.379,A -85,B 0,C 180,E1 -10019.161,E2 -10019.161} C_VEL
LIN {X 0,Y 418.257,Z 136.381,A -85,B 0,C 180,E1 -10022.844,E2 -10022.844} C_VEL
LIN {X 0,Y 418.245,Z 136.387,A -85,B 0,C 180,E1 -10026.239,E2 -10026.239} C_VEL
LIN {X 0,Y 418.25,Z 136.386,A -85,B 0,C 180,E1 -10029.682,E2 -10029.682} C_VEL
LIN {X 0,Y 418.28,Z 136.381,A -85,B 0,C 180,E1 -10032.329,E2 -10032.329} C_VEL
LIN {X 0,Y 418.248,Z 136.383,A -85,B 0,C 180,E1 -10035.111,E2 -10035.111} C_VEL
LIN {X 0,Y 418.253,Z 136.389,A -85,B 0,C 180,E1 -10037.769,E2 -10037.769} C_VEL
LIN {X 0,Y 418.263,Z 136.38,A -85,B 0,C 180,E1 -10040.617,E2 -10040.617} C_VEL
LIN {X 0,Y 418.242,Z 136.386,A -85,B 0,C 180,E1 -10043.976,E2 -10043.976} C_VEL
LIN {X 0,Y 418.254,Z 136.384,A -85,B 0,C 180,E1 -10047.156,E2 -10047.156} C_VEL
LIN {X 0,Y 418.265,Z 136.381,A -85,B 0,C 180,E1 -10050.896,E2 -10050.896} C_VEL
LIN {X 0,Y 418.267,Z 136.381,A -85,B 0,C 180,E1 -10054.096,E2 -10054.096} C_VEL
LIN {X 0,Y 418.235,Z 136.39,A -85,B 0,C 180,E1 -10057.264,E2 -10057.264} C_VEL
LIN {X 0,Y 418.28,Z 136.378,A -85,B 0,C 180,E1 -10060.364,E2 -10060.364} C_VEL
LIN {X 0,Y 418.314,Z 136.379,A -85,B 0,C 180,E1 -10063.405,E2 -10063.405} C_VEL
LIN {X 0,Y 418.344,Z 136.376,A -85,B 0,C 180,E1 -10066.999,E2 -10066.999} C_VEL
LIN {X 0,Y 418.339,Z 136.371,A -85,B 0,C 180,E1 -10070.329,E2 -10070.329} C_VEL
LIN {X 0,Y 418.485,Z 136.357,A -85,B 0,C 180,E1 -10073.249,E2 -10073.249} C_VEL
LIN {X 0,Y 418.337,Z 136.376,A -85,B 0,C 180,E1 -10075.182,E2 -10075.182} C_VEL
LIN {X 0,Y 418.543,Z 136.346,A -85,B 0,C 180,E1 -10078.076,E2 -10078.076} C_VEL
LIN {X 0,Y 418.671,Z 136.33,A -85,B 0,C 180,E1 -10080,E2 -10080} C_VEL
LIN {X 0,Y 418.508,Z 136.356,A -85,B 0,C 180,E1 -10082.888,E2 -10082.888} C_VEL
LIN {X 0,Y 418.493,Z 136.359,A -85,B 0,C 180,E1 -10086.751,E2 -10086.751} C_VEL
LIN {X 0,Y 418.34,Z 136.371,A -85,B 0,C 180,E1 -10089.672,E2 -10089.672} C_VEL
LIN {X 0,Y 418.345,Z 136.373,A -85,B 0,C 180,E1 -10093.001,E2 -10093.001} C_VEL
LIN {X 0,Y 418.312,Z 136.379,A -85,B 0,C 180,E1 -10096.736,E2 -10096.736} C_VEL
LIN {X 0,Y 418.27,Z 136.38,A -85,B 0,C 180,E1 -10099.791,E2 -10099.791} C_VEL
LIN {X 0,Y 418.23,Z 136.387,A -85,B 0,C 180,E1 -10102.737,E2 -10102.737} C_VEL
LIN {X 0,Y 418.267,Z 136.382,A -85,B 0,C 180,E1 -10105.905,E2 -10105.905} C_VEL
LIN {X 0,Y 418.264,Z 136.38,A -85,B 0,C 180,E1 -10109.162,E2 -10109.162} C_VEL
LIN {X 0,Y 418.257,Z 136.382,A -85,B 0,C 180,E1 -10112.844,E2 -10112.844} C_VEL
LIN {X 0,Y 418.247,Z 136.388,A -85,B 0,C 180,E1 -10116.239,E2 -10116.239} C_VEL
LIN {X 0,Y 418.264,Z 136.383,A -85,B 0,C 180,E1 -10119.681,E2 -10119.681} C_VEL
LIN {X 0,Y 418.245,Z 136.386,A -85,B 0,C 180,E1 -10122.324,E2 -10122.324} C_VEL
LIN {X 0,Y 418.237,Z 136.384,A -85,B 0,C 180,E1 -10125.109,E2 -10125.109} C_VEL
LIN {X 0,Y 418.24,Z 136.39,A -85,B 0,C 180,E1 -10127.767,E2 -10127.767} C_VEL
LIN {X 0,Y 418.253,Z 136.382,A -85,B 0,C 180,E1 -10130.62,E2 -10130.62} C_VEL
LIN {X 0,Y 418.244,Z 136.387,A -85,B 0,C 180,E1 -10133.976,E2 -10133.976} C_VEL
LIN {X 0,Y 418.258,Z 136.383,A -85,B 0,C 180,E1 -10137.157,E2 -10137.157} C_VEL
LIN {X 0,Y 418.27,Z 136.382,A -85,B 0,C 180,E1 -10140.896,E2 -10140.896} C_VEL
LIN {X 0,Y 418.334,Z 136.408,A -85,B 0,C 180,E1 -10141.53,E2 -10141.53} C_VEL
LIN {X 0,Y 421.092,Z 150.182,A -85,B 0,C 180,E1 -10144.324,E2 -10144.324} C_VEL
LIN {X 0,Y 421.364,Z 154.177,A -85,B 0,C 180,E1 -10145.093,E2 -10145.093} C_VEL
LIN {X 0,Y 420.301,Z 170.783,A -85,B 0,C 180,E1 -10148.158,E2 -10148.158} C_VEL
LIN {X 0,Y 419.456,Z 185.966,A -85,B 0,C 180,E1 -10150.93,E2 -10150.93} C_VEL
LIN {X 0,Y 419.362,Z 187.468,A -85,B 0,C 180,E1 -10151.204,E2 -10151.204} C_VEL
LIN {X 0,Y 422.994,Z 215.123,A -85,B 0,C 180,E1 -10151.895,E2 -10151.895} C_VEL
LIN {X 0,Y 421.832,Z 296.385,A -85,B 0,C 180,E1 -10153.454,E2 -10153.454} C_VEL
LIN {X 0,Y 421.303,Z 309.918,A -85,B 0,C 180,E1 -10153.899,E2 -10153.899} C_VEL
LIN {X 0,Y 420.773,Z 322.336,A -85,B 0,C 180,E1 -10154.5,E2 -10154.5} C_VEL
LIN {X 0,Y 420.088,Z 333.498,A -85,B 0,C 180,E1 -10155.219,E2 -10155.219} C_VEL
LIN {X 0,Y 419.432,Z 345.167,A -85,B 0,C 180,E1 -10156.186,E2 -10156.186} C_VEL
LIN {X 0,Y 418.888,Z 354.981,A -85,B 0,C 180,E1 -10157.197,E2 -10157.197} C_VEL
LIN {X 0,Y 418.363,Z 364.33,A -85,B 0,C 180,E1 -10158.371,E2 -10158.371} C_VEL
LIN {X 0,Y 417.734,Z 373.642,A -85,B 0,C 180,E1 -10159.826,E2 -10159.826} C_VEL
LIN {X 0,Y 417.442,Z 381.141,A -85,B 0,C 180,E1 -10161.285,E2 -10161.285} C_VEL
LIN {X 0,Y 417.247,Z 387.135,A -85,B 0,C 180,E1 -10162.743,E2 -10162.743} C_VEL
LIN {X 0,Y 417.099,Z 391.827,A -85,B 0,C 180,E1 -10164.198,E2 -10164.198} C_VEL
